C03630=1016.141,-94.892,399.074,165.166,56.508,159.988
C03631=1016.146,-94.643,399.065,165.168,56.502,159.987
C03632=1016.150,-94.393,399.056,165.172,56.496,159.987
C03633=1016.156,-94.143,399.048,165.174,56.489,159.987
C03634=1016.160,-93.893,399.039,165.177,56.484,159.986
C03635=1016.165,-93.643,399.030,165.180,56.477,159.986
C03636=1016.171,-93.394,399.022,165.183,56.472,159.986
C03637=1016.175,-93.144,399.013,165.186,56.465,159.985
C03638=1016.180,-92.894,399.004,165.189,56.459,159.985
C03639=1016.185,-92.644,398.995,165.192,56.453,159.985
C03640=1016.190,-92.394,398.986,165.194,56.446,159.984
C03641=1016.196,-92.144,398.978,165.197,56.441,159.983
C03642=1016.200,-91.894,398.969,165.201,56.434,159.983
C03643=1016.206,-91.645,398.960,165.203,56.428,159.983
C03644=1016.210,-91.395,398.951,165.206,56.422,159.982
C03645=1016.215,-91.145,398.942,165.209,56.416,159.982
C03646=1016.221,-90.896,398.934,165.212,56.409,159.982
C03647=1016.225,-90.646,398.925,165.215,56.403,159.981
C03648=1016.230,-90.396,398.916,165.218,56.397,159.981
C03649=1016.235,-90.146,398.907,165.221,56.391,159.980
C03650=1016.240,-89.896,398.899,165.224,56.385,159.980
C03651=1016.246,-89.647,398.889,165.227,56.379,159.980
C03652=1016.250,-89.397,398.880,165.230,56.372,159.979
C03653=1016.256,-89.147,398.872,165.233,56.366,159.979
C03654=1016.260,-88.897,398.863,165.236,56.359,159.978
///RCONF 1,0,0,0,0,0,0,0,0,0,0,0,0,0,0,0,0,0,0,0,0,0,0,0
C03655=1016.266,-88.647,398.854,165.238,56.354,159.978
C03656=1016.272,-88.398,398.845,165.242,56.347,159.978
C03657=1016.276,-88.148,398.836,165.244,56.341,159.977
C03658=1016.281,-87.898,398.827,165.248,56.335,159.977
C03659=1016.286,-87.648,398.818,165.250,56.328,159.976
C03660=1016.291,-87.398,398.809,165.254,56.322,159.976
C03661=1016.296,-87.149,398.800,165.256,56.316,159.975
C03662=1016.301,-86.899,398.791,165.259,56.309,159.975
C03663=1016.307,-86.650,398.783,165.261,56.303,159.975
C03664=1016.312,-86.399,398.773,165.265,56.297,159.974
C03665=1016.317,-86.120,398.763,165.268,56.290,159.974
C03666=1016.324,-85.839,398.753,165.271,56.283,159.973
C03667=1016.329,-85.559,398.743,165.274,56.275,159.973
C03668=1016.334,-85.278,398.733,165.278,56.268,159.972
C03669=1016.340,-85.029,398.724,165.281,56.262,159.972
C03670=1016.345,-84.779,398.714,165.284,56.256,159.972
C03671=1016.350,-84.530,398.706,165.287,56.250,159.971
C03672=1016.355,-84.280,398.697,165.290,56.243,159.971
C03673=1016.361,-84.030,398.687,165.293,56.237,159.970
C03674=1016.366,-83.780,398.679,165.296,56.230,159.970
C03675=1016.370,-83.530,398.670,165.298,56.224,159.969
C03676=1016.376,-83.281,398.661,165.301,56.218,159.969
C03677=1016.381,-83.031,398.652,165.305,56.211,159.969
C03678=1016.386,-82.780,398.643,165.307,56.205,159.968
C03679=1016.392,-82.531,398.633,165.310,56.198,159.968
C03680=1016.396,-82.281,398.624,165.313,56.193,159.967
C03681=1016.402,-82.032,398.615,165.316,56.186,159.967
C03682=1016.407,-81.782,398.606,165.319,56.179,159.966
C03683=1016.412,-81.532,398.597,165.322,56.173,159.966
C03684=1016.417,-81.282,398.587,165.325,56.166,159.965
C03685=1016.422,-81.033,398.579,165.328,56.160,159.965
C03686=1016.429,-80.783,398.569,165.331,56.154,159.965
C03687=1016.433,-80.533,398.560,165.334,56.147,159.964
C03688=1016.438,-80.283,398.552,165.337,56.141,159.964
C03689=1016.443,-80.034,398.542,165.340,56.134,159.963
C03690=1016.449,-79.784,398.532,165.343,56.128,159.963
C03691=1016.454,-79.534,398.523,165.346,56.122,159.962
C03692=1016.459,-79.285,398.514,165.348,56.116,159.962
C03693=1016.464,-79.034,398.504,165.352,56.109,159.962
C03694=1016.469,-78.784,398.494,165.354,56.103,159.961
C03695=1016.474,-78.535,398.485,165.357,56.096,159.961
C03696=1016.479,-78.285,398.476,165.360,56.091,159.960
C03697=1016.484,-78.035,398.466,165.364,56.085,159.960
C03698=1016.490,-77.786,398.457,165.366,56.078,159.959
C03699=1016.494,-77.536,398.448,165.370,56.072,159.959
C03700=1016.500,-77.286,398.437,165.372,56.066,159.959
C03701=1016.505,-77.037,398.428,165.375,56.059,159.958
C03702=1016.510,-76.787,398.419,165.378,56.053,159.958
C03703=1016.515,-76.537,398.409,165.381,56.046,159.957
C03704=1016.520,-76.287,398.399,165.383,56.040,159.957
C03705=1016.525,-76.038,398.391,165.387,56.034,159.956
C03706=1016.531,-75.787,398.381,165.389,56.028,159.956
C03707=1016.536,-75.538,398.371,165.392,56.021,159.955
C03708=1016.541,-75.287,398.361,165.395,56.015,159.955
C03709=1016.546,-75.038,398.352,165.398,56.008,159.955
C03710=1016.551,-74.789,398.342,165.401,56.003,159.954
C03711=1016.557,-74.539,398.332,165.404,55.996,159.954
C03712=1016.561,-74.289,398.323,165.407,55.990,159.953
C03713=1016.567,-74.039,398.313,165.410,55.983,159.953
C03714=1016.571,-73.789,398.303,165.413,55.978,159.952
C03715=1016.576,-73.540,398.293,165.416,55.972,159.952
C03716=1016.582,-73.290,398.283,165.418,55.965,159.952
C03717=1016.587,-73.040,398.273,165.421,55.959,159.951
C03718=1016.592,-72.790,398.263,165.424,55.953,159.951
C03719=1016.597,-72.541,398.253,165.427,55.947,159.950
C03720=1016.602,-72.291,398.243,165.431,55.941,159.950
C03721=1016.607,-72.041,398.233,165.433,55.934,159.949
C03722=1016.612,-71.792,398.224,165.436,55.929,159.949
C03723=1016.617,-71.542,398.213,165.439,55.922,159.949
C03724=1016.622,-71.292,398.204,165.441,55.916,159.948
C03725=1016.628,-71.042,398.194,165.445,55.910,159.948
C03726=1016.632,-70.793,398.184,165.447,55.904,159.947
C03727=1016.638,-70.543,398.174,165.451,55.897,159.947
C03728=1016.643,-70.293,398.164,165.453,55.891,159.946
C03729=1016.649,-70.015,398.153,165.456,55.884,159.946
C03730=1016.654,-69.737,398.141,165.460,55.877,159.945
C03731=1016.660,-69.458,398.130,165.463,55.870,159.945
C03732=1016.665,-69.180,398.120,165.466,55.864,159.944
C03733=1016.671,-68.930,398.110,165.469,55.857,159.944
C03734=1016.676,-68.681,398.100,165.472,55.851,159.944
C03735=1016.681,-68.430,398.090,165.475,55.844,159.943
C03736=1016.686,-68.181,398.080,165.478,55.839,159.943
C03737=1016.692,-67.932,398.069,165.481,55.832,159.942
C03738=1016.697,-67.681,398.059,165.484,55.826,159.942
C03739=1016.702,-67.432,398.049,165.487,55.819,159.941
C03740=1016.707,-67.182,398.039,165.489,55.814,159.941
C03741=1016.712,-66.933,398.029,165.493,55.807,159.941
C03742=1016.717,-66.682,398.018,165.495,55.801,159.940
C03743=1016.722,-66.433,398.008,165.499,55.794,159.940
C03744=1016.727,-66.183,397.998,165.501,55.788,159.939
C03745=1016.732,-65.933,397.988,165.504,55.782,159.939
C03746=1016.738,-65.684,397.978,165.507,55.775,159.938
C03747=1016.743,-65.434,397.967,165.510,55.769,159.938
C03748=1016.748,-65.184,397.958,165.512,55.763,159.937
C03749=1016.753,-64.934,397.947,165.516,55.756,159.937
C03750=1016.758,-64.685,397.938,165.518,55.750,159.936
C03751=1016.764,-64.435,397.928,165.522,55.744,159.936
C03752=1016.769,-64.185,397.917,165.524,55.738,159.935
C03753=1016.774,-63.936,397.907,165.527,55.731,159.935
C03754=1016.780,-63.686,397.897,165.530,55.725,159.934
C03755=1016.784,-63.436,397.887,165.533,55.719,159.934
C03756=1016.790,-63.186,397.877,165.537,55.712,159.934
C03757=1016.796,-62.937,397.866,165.539,55.705,159.933
C03758=1016.800,-62.687,397.856,165.543,55.699,159.933
C03759=1016.806,-62.437,397.846,165.545,55.693,159.932
C03760=1016.811,-62.187,397.836,165.548,55.686,159.932
C03761=1016.816,-61.938,397.825,165.551,55.680,159.931
C03762=1016.822,-61.688,397.815,165.554,55.674,159.931
C03763=1016.827,-61.438,397.805,165.556,55.667,159.930
C03764=1016.831,-61.188,397.795,165.560,55.661,159.930
C03765=1016.837,-60.939,397.784,165.562,55.655,159.929
C03766=1016.843,-60.689,397.773,165.565,55.648,159.929
C03767=1016.847,-60.439,397.764,165.568,55.641,159.928
C03768=1016.853,-60.190,397.753,165.571,55.635,159.928
C03769=1016.859,-59.940,397.743,165.574,55.629,159.927
C03770=1016.863,-59.690,397.733,165.576,55.622,159.927
C03771=1016.869,-59.440,397.723,165.580,55.615,159.926
C03772=1016.875,-59.191,397.712,165.582,55.610,159.926
C03773=1016.880,-58.940,397.702,165.586,55.603,159.925
C03774=1016.885,-58.691,397.692,165.589,55.596,159.925
C03775=1016.891,-58.442,397.681,165.591,55.590,159.924
C03776=1016.896,-58.191,397.671,165.595,55.584,159.924
C03777=1016.902,-57.942,397.660,165.597,55.577,159.923
C03778=1016.907,-57.693,397.650,165.600,55.570,159.923
C03779=1016.912,-57.442,397.640,165.603,55.564,159.922
C03780=1016.918,-57.193,397.629,165.606,55.557,159.922
C03781=1016.922,-56.943,397.618,165.609,55.550,159.921
C03782=1016.928,-56.694,397.608,165.612,55.545,159.921
C03783=1016.933,-56.444,397.598,165.615,55.538,159.920
C03784=1016.938,-56.194,397.588,165.618,55.531,159.920
C03785=1016.944,-55.944,397.577,165.620,55.525,159.919
C03786=1016.950,-55.694,397.566,165.623,55.518,159.919
C03787=1016.955,-55.445,397.556,165.626,55.512,159.918
C03788=1016.960,-55.195,397.546,165.629,55.506,159.918
C03789=1016.966,-54.946,397.535,165.633,55.499,159.917
C03790=1016.971,-54.695,397.525,165.635,55.492,159.917
C03791=1016.977,-54.445,397.515,165.638,55.486,159.916
C03792=1016.982,-54.197,397.504,165.640,55.479,159.915
C03793=1016.988,-53.919,397.492,165.644,55.471,159.915
C03794=1016.995,-53.642,397.480,165.647,55.465,159.914
C03795=1017.000,-53.365,397.469,165.650,55.457,159.914
C03796=1017.006,-53.088,397.457,165.654,55.450,159.913
C03797=1017.012,-52.838,397.447,165.657,55.444,159.913
C03798=1017.017,-52.588,397.436,165.660,55.437,159.912
C03799=1017.022,-52.338,397.425,165.662,55.430,159.912
C03800=1017.027,-52.089,397.415,165.665,55.424,159.911
C03801=1017.033,-51.839,397.404,165.668,55.417,159.911
C03802=1017.038,-51.589,397.394,165.671,55.410,159.910
C03803=1017.044,-51.340,397.383,165.674,55.404,159.909
C03804=1017.050,-51.090,397.373,165.677,55.397,159.909
C03805=1017.055,-50.840,397.362,165.679,55.391,159.908
C03806=1017.060,-50.590,397.351,165.683,55.384,159.908
C03807=1017.065,-50.340,397.339,165.685,55.378,159.907
C03808=1017.071,-50.090,397.329,165.689,55.371,159.907
C03809=1017.076,-49.841,397.318,165.691,55.366,159.906
C03810=1017.081,-49.591,397.307,165.695,55.359,159.906
C03811=1017.086,-49.341,397.295,165.697,55.353,159.905
C03812=1017.092,-49.091,397.285,165.701,55.347,159.905
C03813=1017.097,-48.842,397.275,165.703,55.340,159.904
C03814=1017.102,-48.593,397.263,165.705,55.334,159.904
C03815=1017.108,-48.343,397.252,165.708,55.327,159.903
C03816=1017.113,-48.093,397.241,165.711,55.321,159.903
C03817=1017.119,-47.844,397.230,165.714,55.315,159.902
C03818=1017.123,-47.593,397.219,165.716,55.308,159.902
C03819=1017.129,-47.344,397.208,165.720,55.302,159.901
C03820=1017.134,-47.094,397.197,165.722,55.296,159.901
C03821=1017.140,-46.845,397.186,165.726,55.289,159.900
C03822=1017.145,-46.595,397.174,165.728,55.283,159.900
C03823=1017.150,-46.345,397.163,165.731,55.276,159.899
C03824=1017.155,-46.095,397.152,165.734,55.270,159.899
C03825=1017.161,-45.846,397.141,165.737,55.264,159.898
C03826=1017.166,-45.596,397.130,165.739,55.257,159.898
C03827=1017.172,-45.347,397.119,165.743,55.251,159.897
C03828=1017.177,-45.096,397.108,165.746,55.244,159.897
C03829=1017.182,-44.847,397.097,165.749,55.238,159.896
C03830=1017.187,-44.597,397.086,165.752,55.231,159.896
C03831=1017.193,-44.347,397.075,165.754,55.225,159.895
C03832=1017.198,-44.098,397.063,165.757,55.218,159.895
C03833=1017.204,-43.848,397.052,165.760,55.212,159.894
C03834=1017.209,-43.598,397.041,165.763,55.205,159.893
C03835=1017.215,-43.349,397.030,165.765,55.199,159.893
C03836=1017.220,-43.099,397.019,165.769,55.193,159.893
C03837=1017.225,-42.850,397.008,165.771,55.186,159.892
C03838=1017.230,-42.600,396.996,165.775,55.180,159.891
C03839=1017.236,-42.350,396.985,165.777,55.173,159.891
C03840=1017.241,-42.101,396.974,165.780,55.167,159.890
C03841=1017.247,-41.850,396.963,165.782,55.160,159.890
C03842=1017.252,-41.601,396.951,165.786,55.154,159.889
C03843=1017.258,-41.351,396.940,165.789,55.147,159.889
C03844=1017.263,-41.101,396.929,165.791,55.140,159.888
C03845=1017.269,-40.852,396.918,165.794,55.134,159.887
C03846=1017.274,-40.602,396.907,165.797,55.128,159.887
C03847=1017.280,-40.352,396.896,165.800,55.121,159.887
C03848=1017.285,-40.103,396.884,165.803,55.115,159.886
C03849=1017.291,-39.854,396.873,165.806,55.108,159.885
C03850=1017.296,-39.604,396.861,165.809,55.102,159.885
C03851=1017.301,-39.353,396.849,165.811,55.095,159.884
C03852=1017.307,-39.104,396.838,165.815,55.088,159.884
C03853=1017.312,-38.854,396.827,165.817,55.082,159.883
C03854=1017.317,-38.604,396.815,165.820,55.077,159.883
C03855=1017.322,-38.355,396.803,165.823,55.070,159.882
C03856=1017.328,-38.106,396.792,165.825,55.063,159.881
C03857=1017.334,-37.828,396.779,165.829,55.057,159.881
C03858=1017.339,-37.551,396.767,165.831,55.049,159.880
C03859=1017.346,-37.275,396.754,165.835,55.043,159.880
C03860=1017.351,-36.998,396.741,165.838,55.035,159.879
C03861=1017.356,-36.748,396.730,165.841,55.028,159.879
C03862=1017.362,-36.499,396.717,165.843,55.023,159.878
C03863=1017.368,-36.249,396.706,165.847,55.016,159.878
C03864=1017.373,-35.999,396.695,165.849,55.010,159.877
C03865=1017.378,-35.750,396.682,165.852,55.003,159.876
C03866=1017.383,-35.500,396.671,165.855,54.997,159.876
C03867=1017.389,-35.250,396.659,165.858,54.990,159.875
C03868=1017.395,-35.001,396.648,165.860,54.984,159.875
C03869=1017.400,-34.751,396.636,165.864,54.978,159.874
C03870=1017.405,-34.501,396.625,165.866,54.971,159.874
C03871=1017.410,-34.252,396.612,165.870,54.965,159.873
C03872=1017.416,-34.002,396.601,165.872,54.958,159.873
C03873=1017.422,-33.752,396.590,165.875,54.952,159.872
C03874=1017.427,-33.503,396.578,165.877,54.945,159.871
C03875=1017.432,-33.253,396.566,165.881,54.939,159.871
C03876=1017.438,-33.003,396.554,165.883,54.932,159.870
C03877=1017.443,-32.753,396.542,165.886,54.925,159.870
C03878=1017.449,-32.504,396.531,165.888,54.919,159.869
C03879=1017.454,-32.255,396.519,165.892,54.912,159.869
C03880=1017.459,-32.004,396.507,165.895,54.907,159.868
C03881=1017.465,-31.755,396.495,165.898,54.900,159.868
C03882=1017.470,-31.505,396.483,165.900,54.894,159.867
C03883=1017.476,-31.256,396.472,165.903,54.887,159.867
C03884=1017.481,-31.006,396.460,165.906,54.881,159.866
C03885=1017.486,-30.756,396.449,165.909,54.874,159.865
C03886=1017.492,-30.507,396.436,165.911,54.868,159.865
C03887=1017.497,-30.256,396.425,165.915,54.861,159.864
C03888=1017.503,-30.008,396.413,165.917,54.855,159.864
C03889=1017.508,-29.758,396.401,165.920,54.848,159.863
C03890=1017.514,-29.508,396.389,165.923,54.842,159.862
C03891=1017.519,-29.258,396.377,165.926,54.835,159.862
C03892=1017.525,-29.009,396.365,165.928,54.829,159.861
C03893=1017.531,-28.759,396.354,165.931,54.822,159.861
C03894=1017.536,-28.510,396.342,165.935,54.815,159.860
C03895=1017.541,-28.260,396.330,165.937,54.809,159.860
C03896=1017.547,-28.010,396.318,165.940,54.802,159.859
C03897=1017.552,-27.760,396.306,165.942,54.795,159.858
C03898=1017.557,-27.511,396.294,165.946,54.789,159.858
C03899=1017.563,-27.261,396.282,165.948,54.783,159.857
C03900=1017.568,-27.011,396.270,165.951,54.777,159.857
C03901=1017.574,-26.762,396.258,165.954,54.770,159.856
C03902=1017.580,-26.512,396.245,165.956,54.764,159.855
C03903=1017.585,-26.262,396.234,165.959,54.757,159.855
C03904=1017.591,-26.012,396.221,165.962,54.751,159.854
C03905=1017.596,-25.763,396.209,165.965,54.744,159.854
C03906=1017.601,-25.514,396.197,165.968,54.739,159.853
C03907=1017.607,-25.264,396.185,165.970,54.732,159.853
C03908=1017.611,-25.014,396.172,165.973,54.726,159.852
C03909=1017.617,-24.764,396.160,165.976,54.719,159.852
C03910=1017.623,-24.515,396.148,165.979,54.713,159.851
C03911=1017.628,-24.265,396.136,165.981,54.706,159.850
C03912=1017.633,-24.015,396.124,165.985,54.700,159.850
C03913=1017.639,-23.766,396.111,165.987,54.693,159.849
C03914=1017.645,-23.516,396.099,165.989,54.687,159.849
C03915=1017.650,-23.266,396.087,165.993,54.680,159.848
C03916=1017.655,-23.017,396.075,165.995,54.674,159.847
C03917=1017.661,-22.767,396.063,165.998,54.667,159.847
C03918=1017.666,-22.518,396.050,166.001,54.661,159.846
C03919=1017.671,-22.268,396.037,166.004,54.654,159.846
C03920=1017.676,-22.018,396.026,166.006,54.648,159.845
C03921=1017.683,-21.741,396.012,166.010,54.641,159.845
C03922=1017.689,-21.463,395.999,166.012,54.634,159.844
C03923=1017.695,-21.185,395.985,166.015,54.627,159.843
C03924=1017.701,-20.907,395.971,166.019,54.620,159.843
C03925=1017.707,-20.658,395.959,166.022,54.613,159.842
C03926=1017.713,-20.408,395.946,166.024,54.606,159.841
C03927=1017.718,-20.158,395.935,166.027,54.600,159.841
C03928=1017.724,-19.908,395.922,166.029,54.593,159.840
C03929=1017.728,-19.659,395.909,166.033,54.587,159.840
C03930=1017.734,-19.409,395.897,166.035,54.580,159.839
C03931=1017.739,-19.160,395.884,166.038,54.574,159.838
C03932=1017.745,-18.910,395.872,166.041,54.567,159.838
C03933=1017.751,-18.661,395.860,166.044,54.561,159.837
C03934=1017.756,-18.411,395.847,166.046,54.555,159.837
C03935=1017.762,-18.162,395.835,166.050,54.548,159.836
C03936=1017.768,-17.912,395.822,166.052,54.542,159.835
C03937=1017.773,-17.663,395.810,166.055,54.535,159.835
C03938=1017.778,-17.412,395.798,166.058,54.529,159.834
C03939=1017.783,-17.163,395.786,166.061,54.522,159.834
C03940=1017.789,-16.913,395.773,166.063,54.515,159.833
C03941=1017.795,-16.663,395.760,166.066,54.508,159.832
C03942=1017.800,-16.414,395.748,166.069,54.502,159.832
C03943=1017.806,-16.164,395.736,166.072,54.495,159.831
C03944=1017.811,-15.915,395.724,166.074,54.489,159.830
C03945=1017.817,-15.665,395.710,166.078,54.482,159.830
C03946=1017.822,-15.416,395.698,166.080,54.476,159.829
C03947=1017.828,-15.166,395.685,166.082,54.470,159.829
C03948=1017.833,-14.917,395.672,166.086,54.463,159.828
C03949=1017.839,-14.667,395.660,166.088,54.457,159.827
C03950=1017.844,-14.417,395.646,166.090,54.451,159.827
C03951=1017.849,-14.167,395.634,166.094,54.444,159.826
C03952=1017.855,-13.917,395.622,166.096,54.438,159.826
C03953=1017.860,-13.669,395.608,166.099,54.431,159.825
C03954=1017.866,-13.419,395.596,166.102,54.425,159.824
C03955=1017.871,-13.168,395.583,166.104,54.419,159.824
C03956=1017.876,-12.919,395.570,166.107,54.412,159.823
C03957=1017.882,-12.669,395.558,166.110,54.406,159.823
C03958=1017.888,-12.420,395.544,166.113,54.399,159.822
C03959=1017.893,-12.171,395.532,166.115,54.393,159.821
C03960=1017.898,-11.920,395.519,166.118,54.387,159.821
C03961=1017.903,-11.671,395.506,166.121,54.380,159.820
C03962=1017.909,-11.421,395.494,166.123,54.374,159.820
C03963=1017.915,-11.172,395.480,166.127,54.367,159.819
C03964=1017.920,-10.923,395.468,166.129,54.361,159.818
C03965=1017.926,-10.673,395.455,166.132,54.355,159.818
C03966=1017.931,-10.423,395.442,166.135,54.348,159.817
C03967=1017.937,-10.174,395.429,166.137,54.342,159.817
C03968=1017.942,-9.924,395.416,166.141,54.335,159.816
C03969=1017.948,-9.674,395.403,166.143,54.329,159.815
C03970=1017.954,-9.425,395.391,166.146,54.321,159.815
C03971=1017.959,-9.175,395.377,166.148,54.315,159.814
C03972=1017.965,-8.925,395.365,166.151,54.309,159.813
C03973=1017.969,-8.676,395.352,166.154,54.302,159.813
C03974=1017.975,-8.427,395.339,166.156,54.296,159.812
C03975=1017.981,-8.177,395.326,166.160,54.289,159.812
C03976=1017.986,-7.926,395.313,166.162,54.283,159.811
C03977=1017.992,-7.678,395.300,166.165,54.277,159.811
C03978=1017.997,-7.428,395.287,166.167,54.270,159.810
C03979=1018.003,-7.178,395.275,166.171,54.263,159.809
C03980=1018.009,-6.929,395.262,166.173,54.257,159.808
C03981=1018.014,-6.679,395.248,166.175,54.251,159.808
C03982=1018.020,-6.429,395.236,166.179,54.244,159.807
C03983=1018.025,-6.180,395.222,166.181,54.238,159.807
C03984=1018.031,-5.930,395.210,166.184,54.230,159.806
C03985=1018.038,-5.650,395.195,166.187,54.223,159.805
C03986=1018.043,-5.371,395.180,166.190,54.216,159.804
C03987=1018.050,-5.091,395.166,166.193,54.209,159.804
C03988=1018.056,-4.812,395.151,166.196,54.202,159.803
C03989=1018.062,-4.562,395.138,166.199,54.194,159.802
C03990=1018.067,-4.313,395.125,166.201,54.188,159.802
C03991=1018.072,-4.063,395.112,166.204,54.182,159.801
C03992=1018.078,-3.813,395.098,166.207,54.175,159.801
C03993=1018.083,-3.563,395.085,166.210,54.169,159.800
C03994=1018.089,-3.314,395.072,166.212,54.163,159.799
C03995=1018.094,-3.064,395.059,166.215,54.156,159.799
C03996=1018.099,-2.815,395.045,166.218,54.150,159.798
C03997=1018.105,-2.565,395.031,166.220,54.144,159.797
C03998=1018.111,-2.315,395.019,166.223,54.137,159.797
C03999=1018.116,-2.066,395.005,166.226,54.131,159.796
C04000=1018.121,-1.817,394.991,166.228,54.125,159.796
C04001=1018.126,-1.567,394.978,166.232,54.118,159.795
C04002=1018.132,-1.317,394.964,166.234,54.112,159.794
C04003=1018.138,-1.068,394.951,166.236,54.106,159.794
C04004=1018.143,-0.818,394.938,166.239,54.099,159.793
C04005=1018.148,-0.569,394.924,166.242,54.093,159.793
C04006=1018.153,-0.319,394.911,166.244,54.087,159.792
C04007=1018.159,-0.069,394.898,166.247,54.080,159.791
C04008=1018.165,0.180,394.884,166.250,54.074,159.791
C04009=1018.170,0.430,394.870,166.253,54.068,159.790
C04010=1018.175,0.680,394.857,166.255,54.061,159.789
C04011=1018.180,0.929,394.844,166.258,54.055,159.789
C04012=1018.186,1.178,394.830,166.261,54.049,159.788
C04013=1018.192,1.428,394.817,166.263,54.042,159.788
C04014=1018.197,1.678,394.803,166.266,54.035,159.787
C04015=1018.203,1.927,394.789,166.268,54.029,159.786
C04016=1018.209,2.177,394.776,166.272,54.022,159.786
C04017=1018.214,2.426,394.762,166.274,54.016,159.785
C04018=1018.219,2.676,394.749,166.277,54.010,159.784
C04019=1018.224,2.925,394.736,166.280,54.003,159.784
C04020=1018.230,3.175,394.722,166.282,53.997,159.783
C04021=1018.236,3.424,394.709,166.285,53.991,159.783
C04022=1018.241,3.674,394.695,166.288,53.983,159.782
C04023=1018.247,3.924,394.682,166.290,53.977,159.781
C04024=1018.252,4.174,394.668,166.292,53.971,159.780
C04025=1018.258,4.423,394.654,166.296,53.964,159.780
C04026=1018.264,4.672,394.641,166.298,53.958,159.779
C04027=1018.269,4.922,394.627,166.301,53.952,159.779
C04028=1018.274,5.172,394.614,166.304,53.945,159.778
C04029=1018.280,5.422,394.600,166.306,53.939,159.777
C04030=1018.286,5.671,394.586,166.309,53.932,159.777
C04031=1018.292,5.921,394.573,166.312,53.926,159.776
C04032=1018.297,6.169,394.559,166.314,53.920,159.775
C04033=1018.302,6.419,394.545,166.317,53.912,159.775
C04034=1018.307,6.669,394.532,166.320,53.906,159.774
C04035=1018.313,6.918,394.519,166.322,53.900,159.773
C04036=1018.319,7.168,394.505,166.325,53.893,159.773
C04037=1018.324,7.418,394.491,166.327,53.886,159.772
C04038=1018.330,7.667,394.477,166.331,53.880,159.771
C04039=1018.335,7.917,394.463,166.333,53.874,159.771
C04040=1018.342,8.166,394.450,166.336,53.867,159.770
C04041=1018.347,8.416,394.436,166.339,53.860,159.769
C04042=1018.352,8.665,394.422,166.341,53.854,159.769
C04043=1018.358,8.915,394.408,166.344,53.847,159.768
C04044=1018.363,9.165,394.395,166.347,53.841,159.767
C04045=1018.369,9.414,394.382,166.349,53.834,159.767
C04046=1018.375,9.664,394.368,166.352,53.828,159.766
C04047=1018.380,9.913,394.354,166.355,53.821,159.765
C04048=1018.386,10.163,394.340,166.358,53.814,159.765
C04049=1018.393,10.444,394.325,166.361,53.807,159.764
C04050=1018.399,10.726,394.309,166.363,53.800,159.763
C04051=1018.405,11.008,394.294,166.366,53.792,159.762
C04052=1018.411,11.289,394.278,166.369,53.785,159.762
C04053=1018.418,11.538,394.264,166.371,53.778,159.761
C04054=1018.423,11.788,394.251,166.375,53.772,159.760
C04055=1018.429,12.038,394.237,166.377,53.765,159.760
C04056=1018.434,12.287,394.223,166.380,53.758,159.759
C04057=1018.440,12.550,394.209,166.383,53.752,159.758
C04058=1018.446,12.813,394.194,166.386,53.745,159.757
C04059=1018.452,13.076,394.180,166.389,53.737,159.757
C04060=1018.458,13.339,394.165,166.391,53.731,159.756
C04061=1018.463,13.588,394.151,166.394,53.724,159.755
C04062=1018.469,13.838,394.137,166.396,53.718,159.755
C04063=1018.474,14.087,394.122,166.399,53.712,159.754
C04064=1018.480,14.336,394.109,166.402,53.705,159.753
C04065=1018.485,14.586,394.095,166.405,53.699,159.753
C04066=1018.491,14.836,394.081,166.407,53.692,159.752
C04067=1018.496,15.085,394.067,166.410,53.685,159.751
C04068=1018.502,15.335,394.051,166.413,53.679,159.751
C04069=1018.508,15.585,394.038,166.415,53.673,159.750
C04070=1018.513,15.834,394.024,166.418,53.666,159.749
C04071=1018.518,16.084,394.010,166.420,53.660,159.749
C04072=1018.524,16.333,393.995,166.423,53.654,159.748
C04073=1018.530,16.582,393.981,166.425,53.647,159.747
C04074=1018.535,16.832,393.968,166.428,53.640,159.746
C04075=1018.541,17.082,393.954,166.431,53.634,159.746
C04076=1018.546,17.331,393.939,166.433,53.628,159.745
C04077=1018.553,17.581,393.925,166.437,53.621,159.745
C04078=1018.557,17.831,393.910,166.439,53.614,159.744
C04079=1018.563,18.080,393.897,166.441,53.608,159.743
C04080=1018.569,18.329,393.882,166.444,53.602,159.743
C04081=1018.574,18.579,393.868,166.446,53.595,159.742
C04082=1018.579,18.828,393.854,166.450,53.588,159.741
C04083=1018.586,19.078,393.839,166.452,53.582,159.741
C04084=1018.591,19.328,393.825,166.455,53.576,159.740
C04085=1018.596,19.578,393.811,166.457,53.569,159.739
C04086=1018.602,19.826,393.796,166.460,53.562,159.738
C04087=1018.607,20.076,393.783,166.463,53.556,159.738
C04088=1018.613,20.325,393.768,166.465,53.550,159.737
C04089=1018.618,20.576,393.753,166.468,53.543,159.736
C04090=1018.624,20.825,393.739,166.471,53.537,159.736
C04091=1018.630,21.074,393.725,166.473,53.531,159.735
C04092=1018.635,21.324,393.711,166.475,53.524,159.734
C04093=1018.640,21.573,393.696,166.478,53.517,159.734
C04094=1018.646,21.823,393.681,166.481,53.511,159.733
C04095=1018.652,22.072,393.667,166.483,53.505,159.732
C04096=1018.658,22.322,393.653,166.487,53.498,159.732
C04097=1018.662,22.572,393.639,166.489,53.492,159.731
C04098=1018.668,22.821,393.624,166.491,53.485,159.730
C04099=1018.674,23.071,393.610,166.495,53.479,159.730
C04100=1018.680,23.320,393.595,166.497,53.472,159.729
C04101=1018.685,23.570,393.581,166.499,53.466,159.728
C04102=1018.690,23.819,393.566,166.503,53.459,159.728
C04103=1018.697,24.069,393.552,166.505,53.452,159.727
C04104=1018.702,24.318,393.537,166.507,53.446,159.726
C04105=1018.707,24.568,393.523,166.511,53.440,159.726
C04106=1018.713,24.817,393.508,166.513,53.433,159.725
C04107=1018.719,25.067,393.494,166.515,53.427,159.724
C04108=1018.724,25.316,393.479,166.519,53.420,159.723
C04109=1018.729,25.566,393.465,166.521,53.413,159.723
C04110=1018.735,25.815,393.450,166.523,53.407,159.722
C04111=1018.742,26.064,393.435,166.525,53.401,159.721
C04112=1018.746,26.314,393.421,166.528,53.394,159.721
C04113=1018.752,26.584,393.405,166.532,53.387,159.720
C04114=1018.759,26.854,393.389,166.534,53.381,159.719
C04115=1018.765,27.123,393.374,166.537,53.373,159.718
C04116=1018.771,27.394,393.358,166.540,53.366,159.718
C04117=1018.776,27.643,393.343,166.542,53.359,159.717
C04118=1018.782,27.892,393.329,166.545,53.353,159.716
C04119=1018.787,28.143,393.314,166.548,53.347,159.716
C04120=1018.793,28.392,393.299,166.550,53.341,159.715
C04121=1018.798,28.641,393.284,166.553,53.334,159.714
C04122=1018.804,28.891,393.269,166.555,53.328,159.713
C04123=1018.809,29.140,393.255,166.558,53.321,159.713
C04124=1018.815,29.389,393.240,166.561,53.315,159.712
C04125=1018.820,29.639,393.224,166.563,53.308,159.711
C04126=1018.826,29.888,393.210,166.565,53.302,159.711
C04127=1018.831,30.138,393.195,166.569,53.295,159.710
C04128=1018.837,30.388,393.181,166.571,53.289,159.709
C04129=1018.842,30.637,393.165,166.573,53.282,159.708
C04130=1018.848,30.886,393.151,166.576,53.276,159.708
C04131=1018.853,31.137,393.136,166.579,53.269,159.707
C04132=1018.859,31.386,393.121,166.581,53.263,159.706
C04133=1018.864,31.635,393.106,166.584,53.257,159.706
C04134=1018.871,31.885,393.091,166.587,53.250,159.705
C04135=1018.876,32.134,393.076,166.589,53.244,159.704
C04136=1018.881,32.383,393.062,166.592,53.237,159.704
C04137=1018.887,32.633,393.047,166.594,53.231,159.703
C04138=1018.893,32.882,393.032,166.597,53.224,159.702
C04139=1018.898,33.132,393.017,166.600,53.218,159.702
C04140=1018.903,33.382,393.001,166.602,53.211,159.701
C04141=1018.909,33.631,392.987,166.605,53.205,159.700
C04142=1018.914,33.881,392.972,166.608,53.198,159.699
C04143=1018.920,34.130,392.957,166.610,53.192,159.699
C04144=1018.925,34.379,392.942,166.612,53.186,159.698
C04145=1018.932,34.629,392.927,166.616,53.178,159.697
C04146=1018.937,34.878,392.912,166.618,53.172,159.697
C04147=1018.943,35.128,392.897,166.620,53.166,159.696
C04148=1018.948,35.378,392.883,166.624,53.159,159.695
C04149=1018.954,35.627,392.868,166.626,53.153,159.694
C04150=1018.959,35.877,392.853,166.628,53.146,159.694
C04151=1018.965,36.126,392.838,166.632,53.140,159.693
C04152=1018.971,36.376,392.822,166.634,53.133,159.692
C04153=1018.976,36.625,392.808,166.636,53.127,159.692
C04154=1018.982,36.875,392.792,166.639,53.121,159.691
C04155=1018.987,37.124,392.777,166.642,53.113,159.690
C04156=1018.993,37.374,392.762,166.644,53.107,159.689
C04157=1018.998,37.623,392.746,166.647,53.101,159.689
C04158=1019.004,37.873,392.731,166.649,53.094,159.688
C04159=1019.009,38.122,392.716,166.652,53.088,159.687
C04160=1019.014,38.371,392.701,166.655,53.082,159.687
C04161=1019.020,38.621,392.686,166.657,53.075,159.686
C04162=1019.026,38.870,392.671,166.659,53.069,159.685
C04163=1019.031,39.120,392.655,166.663,53.062,159.685
C04164=1019.036,39.369,392.640,166.665,53.056,159.684
C04165=1019.042,39.619,392.624,166.667,53.050,159.683
C04166=1019.048,39.868,392.609,166.670,53.043,159.682
C04167=1019.054,40.118,392.594,166.673,53.036,159.682
C04168=1019.059,40.367,392.579,166.676,53.030,159.681
C04169=1019.064,40.617,392.563,166.678,53.024,159.680
C04170=1019.070,40.866,392.548,166.680,53.017,159.679
C04171=1019.076,41.116,392.533,166.684,53.011,159.679
C04172=1019.081,41.365,392.518,166.686,53.004,159.678
C04173=1019.087,41.615,392.502,166.688,52.998,159.677
C04174=1019.092,41.864,392.486,166.691,52.992,159.677
C04175=1019.098,42.113,392.472,166.694,52.985,159.676
C04176=1019.103,42.363,392.456,166.696,52.979,159.675
C04177=1019.109,42.646,392.438,166.699,52.971,159.675
C04178=1019.115,42.929,392.421,166.703,52.964,159.674
C04179=1019.122,43.212,392.403,166.705,52.957,159.673
C04180=1019.128,43.495,392.385,166.707,52.950,159.672
C04181=1019.133,43.744,392.370,166.710,52.944,159.671
C04182=1019.139,43.994,392.354,166.713,52.937,159.671
C04183=1019.144,44.243,392.338,166.716,52.931,159.670
C04184=1019.150,44.493,392.323,166.718,52.924,159.669
C04185=1019.155,44.742,392.308,166.721,52.918,159.669
C04186=1019.161,44.992,392.291,166.723,52.912,159.668
C04187=1019.166,45.241,392.276,166.726,52.906,159.667
C04188=1019.171,45.491,392.261,166.729,52.899,159.666
C04189=1019.177,45.740,392.245,166.731,52.893,159.666
C04190=1019.182,45.990,392.229,166.734,52.887,159.665
C04191=1019.188,46.239,392.213,166.736,52.880,159.664
C04192=1019.192,46.488,392.197,166.738,52.874,159.664
C04193=1019.198,46.738,392.182,166.742,52.867,159.663
C04194=1019.203,46.987,392.166,166.744,52.861,159.662
C04195=1019.209,47.237,392.150,166.746,52.854,159.661
C04196=1019.214,47.486,392.134,166.749,52.848,159.661
C04197=1019.220,47.736,392.119,166.751,52.842,159.660
C04198=1019.226,47.986,392.103,166.755,52.835,159.659
C04199=1019.231,48.234,392.087,166.757,52.829,159.659
C04200=1019.237,48.484,392.072,166.759,52.822,159.658
C04201=1019.242,48.733,392.056,166.762,52.816,159.657
C04202=1019.248,48.983,392.040,166.764,52.810,159.657
C04203=1019.254,49.232,392.024,166.767,52.803,159.656
C04204=1019.259,49.481,392.009,166.770,52.797,159.655
C04205=1019.264,49.731,391.993,166.773,52.791,159.654
C04206=1019.269,49.980,391.977,166.775,52.784,159.654
C04207=1019.275,50.230,391.961,166.778,52.778,159.653
C04208=1019.281,50.480,391.945,166.780,52.771,159.652
C04209=1019.286,50.729,391.930,166.783,52.765,159.652
C04210=1019.292,50.978,391.914,166.785,52.758,159.651
C04211=1019.297,51.228,391.898,166.788,52.752,159.650
C04212=1019.303,51.477,391.882,166.791,52.746,159.649
C04213=1019.308,51.727,391.867,166.793,52.739,159.649
C04214=1019.314,51.976,391.850,166.796,52.733,159.648
C04215=1019.319,52.226,391.835,166.798,52.726,159.647
C04216=1019.325,52.475,391.819,166.801,52.720,159.646
C04217=1019.330,52.724,391.804,166.804,52.713,159.646
C04218=1019.335,52.974,391.787,166.806,52.707,159.645
C04219=1019.341,53.224,391.771,166.808,52.700,159.644
C04220=1019.347,53.473,391.755,166.812,52.694,159.644
C04221=1019.352,53.722,391.739,166.814,52.688,159.643
C04222=1019.358,53.972,391.724,166.816,52.681,159.642
C04223=1019.364,54.221,391.707,166.819,52.675,159.641
C04224=1019.369,54.470,391.692,166.822,52.668,159.641
C04225=1019.375,54.720,391.676,166.825,52.662,159.640
C04226=1019.381,54.970,391.660,166.827,52.655,159.639
C04227=1019.386,55.218,391.645,166.830,52.648,159.638
C04228=1019.392,55.468,391.628,166.832,52.642,159.638
C04229=1019.397,55.718,391.612,166.835,52.635,159.637
C04230=1019.403,55.967,391.596,166.837,52.629,159.636
C04231=1019.408,56.217,391.581,166.840,52.622,159.635
C04232=1019.414,56.466,391.565,166.843,52.616,159.635
C04233=1019.420,56.715,391.548,166.845,52.609,159.634
C04234=1019.425,56.964,391.533,166.848,52.603,159.633
C04235=1019.431,57.214,391.517,166.851,52.596,159.632
C04236=1019.437,57.463,391.501,166.853,52.590,159.632
C04237=1019.442,57.713,391.485,166.855,52.583,159.631
C04238=1019.448,57.962,391.469,166.859,52.577,159.630
C04239=1019.453,58.212,391.454,166.861,52.570,159.629
C04240=1019.459,58.461,391.437,166.863,52.563,159.628
C04241=1019.465,58.744,391.418,166.866,52.556,159.628
C04242=1019.472,59.027,391.401,166.869,52.548,159.627
C04243=1019.478,59.311,391.382,166.872,52.541,159.626
C04244=1019.484,59.592,391.364,166.875,52.533,159.625
C04245=1019.490,59.842,391.348,166.879,52.527,159.624
C04246=1019.496,60.092,391.333,166.881,52.520,159.624
C04247=1019.502,60.341,391.316,166.883,52.514,159.623
C04248=1019.507,60.591,391.300,166.887,52.507,159.622
C04249=1019.512,60.840,391.284,166.889,52.500,159.621
C04250=1019.518,61.089,391.268,166.891,52.494,159.621
C04251=1019.524,61.339,391.252,166.894,52.487,159.620
C04252=1019.530,61.588,391.236,166.897,52.480,159.619
C04253=1019.536,61.838,391.220,166.899,52.474,159.618
C04254=1019.541,62.087,391.204,166.902,52.467,159.618
C04255=1019.547,62.336,391.188,166.904,52.461,159.617
C04256=1019.553,62.585,391.172,166.907,52.455,159.616
C04257=1019.558,62.836,391.156,166.910,52.448,159.615
C04258=1019.564,63.085,391.139,166.913,52.442,159.615
C04259=1019.570,63.334,391.123,166.915,52.435,159.614
C04260=1019.575,63.584,391.106,166.918,52.429,159.613
C04261=1019.580,63.833,391.090,166.921,52.422,159.612
C04262=1019.586,64.082,391.073,166.923,52.416,159.612
C04263=1019.591,64.332,391.057,166.925,52.409,159.611
C04264=1019.597,64.581,391.041,166.928,52.402,159.610
C04265=1019.603,64.831,391.024,166.931,52.396,159.609
C04266=1019.609,65.080,391.008,166.933,52.389,159.608
C04267=1019.614,65.330,390.991,166.936,52.383,159.608
C04268=1019.619,65.578,390.975,166.938,52.376,159.607
C04269=1019.624,65.828,390.958,166.942,52.370,159.606
C04270=1019.630,66.077,390.942,166.944,52.363,159.606
C04271=1019.636,66.327,390.926,166.947,52.357,159.605
C04272=1019.641,66.576,390.909,166.949,52.351,159.604
C04273=1019.647,66.826,390.893,166.952,52.344,159.603
C04274=1019.653,67.075,390.876,166.955,52.337,159.603
C04275=1019.658,67.324,390.860,166.957,52.331,159.602
C04276=1019.663,67.574,390.843,166.959,52.325,159.601
C04277=1019.669,67.823,390.827,166.963,52.318,159.601
C04278=1019.674,68.073,390.810,166.965,52.312,159.600
C04279=1019.680,68.322,390.794,166.967,52.305,159.599
C04280=1019.686,68.572,390.777,166.970,52.299,159.598
C04281=1019.691,68.821,390.761,166.973,52.292,159.597
C04282=1019.697,69.071,390.744,166.976,52.286,159.597
C04283=1019.702,69.320,390.727,166.978,52.279,159.596
C04284=1019.708,69.570,390.711,166.980,52.273,159.595
C04285=1019.713,69.818,390.693,166.983,52.266,159.594
C04286=1019.718,70.068,390.677,166.986,52.260,159.594
C04287=1019.724,70.317,390.660,166.988,52.253,159.593
C04288=1019.729,70.567,390.643,166.991,52.247,159.592
C04289=1019.735,70.816,390.627,166.993,52.241,159.591
C04290=1019.740,71.066,390.610,166.997,52.234,159.591
C04291=1019.746,71.315,390.593,166.999,52.228,159.590
C04292=1019.752,71.564,390.576,167.002,52.222,159.589
C04293=1019.757,71.814,390.560,167.004,52.215,159.588
C04294=1019.762,72.063,390.543,167.007,52.209,159.588
C04295=1019.768,72.313,390.527,167.010,52.202,159.587
C04296=1019.774,72.562,390.509,167.012,52.196,159.586
C04297=1019.779,72.811,390.492,167.014,52.189,159.585
C04298=1019.785,73.061,390.476,167.018,52.182,159.585
C04299=1019.790,73.311,390.459,167.020,52.176,159.584
C04300=1019.796,73.560,390.441,167.022,52.170,159.583
C04301=1019.802,73.809,390.425,167.025,52.164,159.582
C04302=1019.806,74.058,390.409,167.028,52.156,159.582
C04303=1019.812,74.307,390.392,167.031,52.150,159.581
C04304=1019.818,74.556,390.375,167.033,52.144,159.580
C04305=1019.824,74.840,390.356,167.036,52.136,159.579
C04306=1019.831,75.123,390.337,167.039,52.129,159.578
C04307=1019.837,75.405,390.318,167.042,52.121,159.577
C04308=1019.843,75.688,390.299,167.045,52.114,159.577
C04309=1019.849,75.937,390.281,167.047,52.108,159.576
C04310=1019.854,76.187,390.264,167.051,52.101,159.575
C04311=1019.860,76.436,390.248,167.053,52.095,159.574
C04312=1019.865,76.685,390.230,167.056,52.089,159.574
C04313=1019.870,76.935,390.214,167.059,52.082,159.573
C04314=1019.876,77.184,390.196,167.061,52.075,159.572
C04315=1019.881,77.434,390.179,167.064,52.069,159.571
C04316=1019.886,77.683,390.162,167.066,52.062,159.571
C04317=1019.892,77.932,390.145,167.069,52.056,159.570
C04318=1019.898,78.182,390.128,167.072,52.049,159.569
C04319=1019.903,78.431,390.111,167.075,52.043,159.568
C04320=1019.909,78.681,390.094,167.077,52.037,159.568
C04321=1019.914,78.930,390.076,167.080,52.031,159.567
C04322=1019.919,79.179,390.060,167.083,52.024,159.566
C04323=1019.925,79.428,390.042,167.085,52.018,159.565
C04324=1019.930,79.678,390.025,167.088,52.011,159.565
C04325=1019.936,79.927,390.008,167.090,52.005,159.564
C04326=1019.941,80.176,389.990,167.093,51.998,159.563
C04327=1019.946,80.426,389.973,167.096,51.992,159.563
C04328=1019.952,80.675,389.956,167.098,51.985,159.562
C04329=1019.957,80.924,389.939,167.101,51.979,159.561
C04330=1019.963,81.173,389.921,167.103,51.973,159.560
C04331=1019.968,81.424,389.904,167.107,51.966,159.559
C04332=1019.974,81.673,389.886,167.109,51.960,159.559
C04333=1019.979,81.922,389.870,167.111,51.953,159.558
C04334=1019.985,82.172,389.852,167.114,51.947,159.557
C04335=1019.990,82.421,389.834,167.117,51.940,159.556
C04336=1019.995,82.670,389.818,167.120,51.933,159.556
C04337=1020.002,82.919,389.801,167.122,51.927,159.555
C04338=1020.007,83.169,389.784,167.125,51.920,159.554
C04339=1020.012,83.418,389.766,167.128,51.914,159.553
C04340=1020.018,83.667,389.749,167.130,51.908,159.553
C04341=1020.024,83.917,389.731,167.133,51.901,159.552
C04342=1020.029,84.166,389.714,167.136,51.895,159.551
C04343=1020.035,84.415,389.696,167.138,51.888,159.550
C04344=1020.040,84.665,389.679,167.141,51.882,159.549
C04345=1020.045,84.914,389.662,167.144,51.875,159.549
C04346=1020.051,85.163,389.644,167.147,51.869,159.548
C04347=1020.056,85.413,389.627,167.149,51.862,159.547
C04348=1020.062,85.662,389.610,167.152,51.856,159.546
C04349=1020.068,85.911,389.592,167.155,51.849,159.546
C04350=1020.073,86.161,389.575,167.157,51.842,159.545
C04351=1020.079,86.410,389.558,167.160,51.836,159.544
C04352=1020.084,86.659,389.540,167.163,51.829,159.543
C04353=1020.089,86.909,389.523,167.165,51.823,159.543
C04354=1020.095,87.158,389.506,167.168,51.817,159.542
C04355=1020.101,87.407,389.488,167.171,51.810,159.541
C04356=1020.106,87.657,389.471,167.173,51.803,159.540
C04357=1020.112,87.906,389.453,167.176,51.797,159.540
C04358=1020.117,88.155,389.436,167.179,51.790,159.539
C04359=1020.123,88.404,389.418,167.182,51.784,159.538
C04360=1020.128,88.654,389.401,167.184,51.777,159.537
C04361=1020.134,88.904,389.383,167.188,51.771,159.537
C04362=1020.140,89.153,389.366,167.190,51.764,159.536
C04363=1020.145,89.402,389.348,167.192,51.757,159.535
C04364=1020.151,89.651,389.331,167.195,51.751,159.534
C04365=1020.156,89.901,389.313,167.198,51.744,159.533
C04366=1020.161,90.151,389.295,167.201,51.739,159.533
C04367=1020.167,90.400,389.278,167.203,51.732,159.532
C04368=1020.172,90.649,389.260,167.206,51.726,159.531
C04369=1020.178,90.931,389.240,167.209,51.718,159.530
C04370=1020.184,91.214,389.219,167.212,51.711,159.529
C04371=1020.190,91.497,389.199,167.215,51.704,159.528
C04372=1020.197,91.780,389.179,167.218,51.697,159.528
C04373=1020.202,92.030,389.161,167.221,51.690,159.527
C04374=1020.207,92.279,389.144,167.224,51.684,159.526
C04375=1020.213,92.528,389.126,167.226,51.677,159.525
C04376=1020.219,92.778,389.108,167.228,51.671,159.525
C04377=1020.224,93.027,389.090,167.232,51.664,159.524
C04378=1020.229,93.276,389.073,167.234,51.658,159.523
C04379=1020.235,93.525,389.055,167.237,51.652,159.522
C04380=1020.241,93.775,389.037,167.240,51.645,159.522
C04381=1020.246,94.024,389.019,167.243,51.638,159.521
C04382=1020.251,94.273,389.001,167.245,51.632,159.520
C04383=1020.257,94.522,388.984,167.248,51.626,159.519
C04384=1020.262,94.772,388.965,167.251,51.619,159.519
C04385=1020.268,95.021,388.948,167.254,51.613,159.518
C04386=1020.273,95.270,388.930,167.256,51.606,159.517
C04387=1020.279,95.519,388.913,167.259,51.599,159.516
C04388=1020.284,95.769,388.894,167.262,51.593,159.516
C04389=1020.290,96.018,388.876,167.264,51.587,159.515
C04390=1020.295,96.267,388.858,167.268,51.580,159.514
C04391=1020.301,96.517,388.840,167.270,51.574,159.513
C04392=1020.306,96.766,388.822,167.273,51.567,159.512
C04393=1020.312,97.015,388.804,167.276,51.560,159.512
C04394=1020.317,97.264,388.787,167.278,51.554,159.511
C04395=1020.323,97.514,388.768,167.281,51.548,159.510
C04396=1020.328,97.763,388.751,167.284,51.541,159.509
C04397=1020.334,98.012,388.733,167.286,51.534,159.508
C04398=1020.339,98.262,388.715,167.289,51.528,159.508
C04399=1020.345,98.511,388.697,167.292,51.521,159.507
C04400=1020.350,98.760,388.680,167.295,51.515,159.506
C04401=1020.356,99.010,388.660,167.297,51.508,159.505
C04402=1020.361,99.259,388.643,167.301,51.502,159.505
C04403=1020.367,99.508,388.625,167.303,51.495,159.504
C04404=1020.372,99.758,388.607,167.306,51.489,159.503
C04405=1020.377,100.007,388.589,167.309,51.482,159.502
C04406=1020.383,100.256,388.570,167.311,51.476,159.502
C04407=1020.388,100.506,388.552,167.314,51.470,159.501
C04408=1020.394,100.755,388.534,167.316,51.463,159.500
C04409=1020.399,101.004,388.515,167.320,51.457,159.500
C04410=1020.405,101.253,388.497,167.322,51.450,159.499
C04411=1020.410,101.503,388.479,167.325,51.444,159.498
C04412=1020.415,101.752,388.460,167.329,51.438,159.497
C04413=1020.421,102.001,388.442,167.331,51.431,159.496
C04414=1020.426,102.250,388.424,167.334,51.425,159.496
C04415=1020.432,102.500,388.406,167.337,51.418,159.495
C04416=1020.437,102.749,388.387,167.339,51.412,159.494
C04417=1020.442,102.998,388.369,167.342,51.406,159.493
C04418=1020.448,103.247,388.351,167.344,51.399,159.493
C04419=1020.453,103.497,388.332,167.348,51.392,159.492
C04420=1020.459,103.746,388.314,167.350,51.386,159.491
C04421=1020.464,103.995,388.296,167.353,51.380,159.490
C04422=1020.470,104.244,388.278,167.356,51.373,159.490
C04423=1020.475,104.494,388.260,167.359,51.367,159.489
C04424=1020.480,104.743,388.241,167.361,51.360,159.488
C04425=1020.486,104.993,388.223,167.365,51.354,159.487
C04426=1020.491,105.242,388.204,167.367,51.347,159.487
C04427=1020.497,105.491,388.186,167.369,51.341,159.486
C04428=1020.502,105.741,388.168,167.373,51.335,159.485
C04429=1020.507,105.989,388.149,167.375,51.328,159.484
C04430=1020.513,106.239,388.131,167.378,51.321,159.483
C04431=1020.519,106.488,388.112,167.381,51.315,159.483
C04432=1020.525,106.738,388.094,167.384,51.309,159.482
C04433=1020.530,107.020,388.073,167.387,51.301,159.481
C04434=1020.536,107.303,388.052,167.390,51.294,159.480
C04435=1020.543,107.586,388.031,167.393,51.287,159.479
C04436=1020.549,107.870,388.011,167.397,51.279,159.478
C04437=1020.554,108.118,387.992,167.400,51.273,159.478
C04438=1020.560,108.368,387.974,167.402,51.266,159.477
C04439=1020.565,108.617,387.955,167.405,51.259,159.476
C04440=1020.572,108.866,387.937,167.408,51.253,159.475
C04441=1020.577,109.115,387.918,167.411,51.247,159.475
C04442=1020.582,109.365,387.900,167.414,51.240,159.474
C04443=1020.588,109.614,387.881,167.416,51.233,159.473
C04444=1020.593,109.864,387.863,167.420,51.227,159.472
C04445=1020.598,110.112,387.844,167.422,51.221,159.472
C04446=1020.604,110.362,387.825,167.425,51.214,159.471
C04447=1020.609,110.611,387.807,167.428,51.208,159.470
C04448=1020.615,110.860,387.788,167.431,51.201,159.469
C04449=1020.620,111.109,387.769,167.433,51.195,159.468
C04450=1020.626,111.359,387.750,167.437,51.188,159.468
C04451=1020.631,111.608,387.732,167.439,51.182,159.467
C04452=1020.637,111.858,387.714,167.442,51.175,159.466
C04453=1020.642,112.106,387.695,167.445,51.169,159.466
C04454=1020.648,112.356,387.675,167.448,51.163,159.465
C04455=1020.653,112.605,387.657,167.450,51.156,159.464
C04456=1020.658,112.855,387.638,167.454,51.150,159.463
C04457=1020.663,113.103,387.619,167.456,51.143,159.462
C04458=1020.669,113.353,387.600,167.459,51.137,159.462
C04459=1020.674,113.601,387.581,167.462,51.131,159.461
C04460=1020.680,113.851,387.562,167.465,51.125,159.460
C04461=1020.684,114.100,387.544,167.467,51.118,159.459
C04462=1020.690,114.350,387.524,167.471,51.112,159.459
C04463=1020.694,114.599,387.505,167.474,51.105,159.458
C04464=1020.700,114.848,387.486,167.476,51.100,159.457
C04465=1020.705,115.097,387.467,167.479,51.093,159.456
C04466=1020.711,115.346,387.448,167.482,51.087,159.456
C04467=1020.716,115.595,387.429,167.485,51.080,159.455
C04468=1020.721,115.845,387.410,167.488,51.074,159.454
C04469=1020.727,116.095,387.391,167.491,51.068,159.454
C04470=1020.732,116.343,387.372,167.493,51.061,159.453
C04471=1020.738,116.593,387.353,167.496,51.055,159.452
C04472=1020.743,116.841,387.334,167.500,51.048,159.451
C04473=1020.749,117.091,387.315,167.502,51.042,159.451
C04474=1020.754,117.340,387.296,167.505,51.036,159.450
C04475=1020.759,117.589,387.277,167.508,51.029,159.449
C04476=1020.764,117.839,387.257,167.511,51.023,159.448
C04477=1020.769,118.088,387.238,167.513,51.017,159.447
C04478=1020.775,118.338,387.219,167.517,51.011,159.447
C04479=1020.780,118.586,387.200,167.519,51.004,159.446
C04480=1020.786,118.836,387.181,167.523,50.997,159.445
C04481=1020.791,119.085,387.162,167.525,50.991,159.445
C04482=1020.796,119.334,387.143,167.528,50.985,159.444
C04483=1020.802,119.583,387.124,167.532,50.979,159.443
C04484=1020.807,119.832,387.105,167.534,50.972,159.442
C04485=1020.813,120.081,387.086,167.536,50.966,159.441
C04486=1020.819,120.331,387.066,167.540,50.959,159.441
C04487=1020.824,120.580,387.048,167.543,50.953,159.440
C04488=1020.829,120.829,387.028,167.546,50.946,159.439
C04489=1020.834,121.079,387.009,167.549,50.940,159.439
C04490=1020.839,121.328,386.990,167.551,50.934,159.438
C04491=1020.845,121.577,386.970,167.555,50.927,159.437
C04492=1020.851,121.826,386.951,167.557,50.921,159.436
C04493=1020.856,122.075,386.932,167.561,50.914,159.436
C04494=1020.861,122.325,386.913,167.564,50.908,159.435
C04495=1020.867,122.574,386.894,167.566,50.902,159.434
C04496=1020.873,122.822,386.874,167.569,50.895,159.433
C04497=1020.878,123.106,386.853,167.573,50.888,159.432
C04498=1020.884,123.389,386.831,167.576,50.881,159.432
C04499=1020.891,123.672,386.809,167.579,50.874,159.431
C04500=1020.897,123.955,386.787,167.583,50.866,159.430
C04501=1020.903,124.203,386.768,167.586,50.859,159.429
C04502=1020.908,124.452,386.748,167.588,50.853,159.428
C04503=1020.913,124.702,386.729,167.592,50.847,159.428
C04504=1020.919,124.952,386.709,167.594,50.840,159.427
C04505=1020.924,125.200,386.691,167.598,50.833,159.426
C04506=1020.930,125.450,386.671,167.600,50.827,159.425
C04507=1020.936,125.699,386.652,167.604,50.821,159.425
C04508=1020.941,125.948,386.633,167.606,50.814,159.424
C04509=1020.947,126.197,386.613,167.610,50.808,159.423
C04510=1020.952,126.446,386.594,167.612,50.801,159.422
C04511=1020.958,126.696,386.575,167.616,50.795,159.421
C04512=1020.963,126.944,386.556,167.619,50.789,159.421
C04513=1020.968,127.194,386.536,167.622,50.782,159.420
C04514=1020.974,127.444,386.517,167.625,50.775,159.419
C04515=1020.980,127.692,386.497,167.628,50.769,159.418
C04516=1020.985,127.942,386.478,167.631,50.763,159.418
C04517=1020.991,128.191,386.459,167.634,50.756,159.417
C04518=1020.996,128.440,386.439,167.637,50.750,159.416
C04519=1021.002,128.689,386.420,167.640,50.743,159.415
C04520=1021.008,128.938,386.400,167.643,50.737,159.415
C04521=1021.013,129.187,386.381,167.646,50.730,159.414
C04522=1021.018,129.437,386.362,167.649,50.724,159.413
C04523=1021.024,129.686,386.342,167.652,50.717,159.412
C04524=1021.030,129.935,386.322,167.655,50.711,159.412
C04525=1021.035,130.184,386.303,167.657,50.704,159.411
C04526=1021.040,130.433,386.284,167.661,50.698,159.410
C04527=1021.046,130.682,386.264,167.664,50.692,159.409
C04528=1021.051,130.932,386.244,167.667,50.685,159.409
C04529=1021.057,131.181,386.224,167.670,50.679,159.408
C04530=1021.062,131.430,386.205,167.673,50.672,159.407
C04531=1021.067,131.679,386.184,167.676,50.667,159.406
C04532=1021.073,131.928,386.165,167.680,50.660,159.406
C04533=1021.078,132.177,386.145,167.682,50.654,159.405
C04534=1021.084,132.427,386.125,167.685,50.648,159.404
C04535=1021.089,132.676,386.106,167.688,50.641,159.403
C04536=1021.094,132.924,386.086,167.691,50.635,159.403
C04537=1021.099,133.174,386.066,167.695,50.628,159.402
C04538=1021.105,133.423,386.046,167.697,50.622,159.401
C04539=1021.110,133.673,386.026,167.701,50.616,159.401
C04540=1021.116,133.922,386.006,167.703,50.609,159.400
C04541=1021.121,134.171,385.987,167.707,50.603,159.399
C04542=1021.127,134.420,385.967,167.710,50.596,159.398
C04543=1021.132,134.669,385.948,167.713,50.590,159.398
C04544=1021.137,134.918,385.927,167.716,50.584,159.397
C04545=1021.143,135.167,385.907,167.719,50.577,159.396
C04546=1021.148,135.417,385.887,167.722,50.571,159.395
C04547=1021.154,135.665,385.867,167.726,50.565,159.395
C04548=1021.159,135.915,385.848,167.728,50.558,159.394
C04549=1021.165,136.164,385.828,167.732,50.552,159.393
C04550=1021.170,136.414,385.808,167.734,50.545,159.392
C04551=1021.175,136.662,385.788,167.737,50.540,159.392
C04552=1021.181,136.911,385.768,167.741,50.533,159.391
C04553=1021.186,137.160,385.748,167.743,50.527,159.390
C04554=1021.192,137.409,385.728,167.747,50.520,159.389
C04555=1021.197,137.659,385.707,167.749,50.514,159.389
C04556=1021.202,137.908,385.688,167.753,50.508,159.388
C04557=1021.208,138.157,385.667,167.756,50.501,159.387
C04558=1021.214,138.406,385.647,167.759,50.495,159.387
C04559=1021.219,138.656,385.628,167.762,50.489,159.386
C04560=1021.224,138.905,385.607,167.766,50.483,159.385
C04561=1021.230,139.187,385.584,167.769,50.475,159.384
C04562=1021.236,139.470,385.561,167.772,50.468,159.383
C04563=1021.242,139.753,385.539,167.776,50.461,159.383
C04564=1021.248,140.036,385.516,167.780,50.454,159.382
C04565=1021.254,140.285,385.496,167.782,50.447,159.381
C04566=1021.259,140.534,385.475,167.786,50.441,159.380
C04567=1021.264,140.783,385.454,167.789,50.435,159.380
C04568=1021.269,141.033,385.435,167.793,50.429,159.379
C04569=1021.275,141.282,385.415,167.795,50.422,159.378
C04570=1021.280,141.531,385.394,167.799,50.416,159.378
C04571=1021.286,141.780,385.374,167.801,50.410,159.377
C04572=1021.291,142.029,385.353,167.805,50.404,159.376
C04573=1021.297,142.278,385.333,167.808,50.397,159.375
C04574=1021.302,142.528,385.313,167.812,50.391,159.375
C04575=1021.307,142.777,385.293,167.814,50.385,159.374
C04576=1021.313,143.026,385.273,167.818,50.379,159.373
C04577=1021.318,143.275,385.252,167.820,50.372,159.372
C04578=1021.324,143.524,385.232,167.824,50.365,159.372
C04579=1021.329,143.773,385.211,167.827,50.360,159.371
C04580=1021.335,144.022,385.191,167.830,50.353,159.370
C04581=1021.340,144.271,385.171,167.834,50.347,159.370
C04582=1021.345,144.520,385.150,167.837,50.340,159.369
C04583=1021.351,144.769,385.129,167.840,50.334,159.368
C04584=1021.356,145.019,385.110,167.843,50.328,159.367
C04585=1021.362,145.268,385.090,167.846,50.321,159.367
C04586=1021.367,145.517,385.069,167.849,50.315,159.366
C04587=1021.372,145.766,385.049,167.853,50.309,159.365
C04588=1021.378,146.015,385.029,167.856,50.303,159.364
C04589=1021.383,146.264,385.008,167.859,50.296,159.364
C04590=1021.389,146.513,384.987,167.863,50.290,159.363
C04591=1021.394,146.762,384.967,167.865,50.284,159.362
C04592=1021.399,147.011,384.946,167.869,50.278,159.362
C04593=1021.405,147.260,384.925,167.872,50.271,159.361
C04594=1021.411,147.510,384.904,167.876,50.265,159.360
C04595=1021.416,147.759,384.884,167.878,50.259,159.359
C04596=1021.421,148.008,384.863,167.882,50.253,159.359
C04597=1021.426,148.257,384.843,167.885,50.247,159.358
C04598=1021.432,148.506,384.822,167.888,50.240,159.357
C04599=1021.437,148.755,384.801,167.891,50.234,159.357
C04600=1021.442,149.004,384.781,167.895,50.228,159.356
C04601=1021.448,149.253,384.760,167.898,50.222,159.355
C04602=1021.453,149.502,384.739,167.901,50.215,159.355
C04603=1021.458,149.751,384.718,167.905,50.209,159.354
C04604=1021.463,150.000,384.698,167.908,50.203,159.353
C04605=1021.469,150.250,384.677,167.911,50.197,159.353
C04606=1021.475,150.498,384.656,167.914,50.190,159.352
C04607=1021.480,150.748,384.635,167.918,50.184,159.351
C04608=1021.485,150.997,384.615,167.920,50.178,159.350
C04609=1021.491,151.246,384.594,167.924,50.172,159.350
C04610=1021.496,151.495,384.574,167.928,50.165,159.349
C04611=1021.501,151.743,384.552,167.931,50.159,159.348
C04612=1021.507,151.993,384.532,167.935,50.153,159.348
C04613=1021.513,152.242,384.511,167.937,50.147,159.347
C04614=1021.518,152.492,384.490,167.941,50.141,159.346
C04615=1021.523,152.740,384.469,167.944,50.134,159.345
C04616=1021.529,152.989,384.448,167.947,50.128,159.345
C04617=1021.534,153.238,384.428,167.951,50.122,159.344
C04618=1021.539,153.487,384.407,167.954,50.116,159.343
C04619=1021.545,153.737,384.386,167.957,50.109,159.343
C04620=1021.551,153.986,384.365,167.960,50.104,159.342
C04621=1021.555,154.235,384.343,167.964,50.097,159.341
C04622=1021.561,154.484,384.323,167.968,50.091,159.341
C04623=1021.566,154.732,384.301,167.970,50.085,159.340
C04624=1021.572,154.982,384.280,167.974,50.078,159.339
C04625=1021.578,155.264,384.257,167.977,50.072,159.338
C04626=1021.584,155.547,384.233,167.982,50.065,159.338
C04627=1021.590,155.829,384.209,167.985,50.057,159.337
C04628=1021.596,156.113,384.185,167.989,50.050,159.336
C04629=1021.601,156.361,384.164,167.993,50.044,159.335
C04630=1021.607,156.610,384.143,167.996,50.038,159.335
C04631=1021.613,156.860,384.122,167.999,50.032,159.334
C04632=1021.617,157.109,384.101,168.003,50.026,159.333
C04633=1021.623,157.357,384.079,168.006,50.020,159.332
C04634=1021.628,157.607,384.059,168.009,50.014,159.332
C04635=1021.634,157.855,384.038,168.013,50.007,159.331
C04636=1021.640,158.105,384.017,168.016,50.001,159.330
C04637=1021.645,158.353,383.995,168.019,49.994,159.330
C04638=1021.650,158.603,383.974,168.023,49.988,159.329
C04639=1021.656,158.852,383.953,168.026,49.983,159.328
C04640=1021.661,159.101,383.932,168.030,49.976,159.328
C04641=1021.666,159.350,383.910,168.033,49.970,159.327
C04642=1021.672,159.599,383.889,168.037,49.964,159.326
C04643=1021.677,159.848,383.867,168.039,49.959,159.326
C04644=1021.681,160.097,383.846,168.043,49.952,159.325
C04645=1021.687,160.346,383.824,168.047,49.946,159.324
C04646=1021.692,160.595,383.802,168.050,49.940,159.324
C04647=1021.697,160.844,383.780,168.054,49.934,159.323
C04648=1021.703,161.093,383.759,168.057,49.929,159.322
C04649=1021.707,161.342,383.738,168.061,49.923,159.322
C04650=1021.712,161.591,383.716,168.063,49.916,159.321
C04651=1021.718,161.840,383.694,168.067,49.910,159.320
C04652=1021.723,162.089,383.672,168.071,49.904,159.320
C04653=1021.729,162.338,383.651,168.074,49.899,159.319
C04654=1021.734,162.586,383.629,168.078,49.893,159.319
C04655=1021.739,162.837,383.608,168.080,49.886,159.318
C04656=1021.744,163.085,383.586,168.084,49.880,159.317
C04657=1021.749,163.334,383.565,168.088,49.874,159.317
C04658=1021.755,163.583,383.542,168.091,49.868,159.316
C04659=1021.760,163.832,383.521,168.095,49.862,159.315
C04660=1021.765,164.081,383.499,168.098,49.856,159.314
C04661=1021.770,164.330,383.477,168.102,49.850,159.314
C04662=1021.776,164.579,383.456,168.105,49.844,159.313
C04663=1021.780,164.828,383.435,168.108,49.838,159.313
C04664=1021.787,165.077,383.413,168.112,49.832,159.312
C04665=1021.791,165.326,383.391,168.116,49.826,159.311
C04666=1021.796,165.575,383.369,168.119,49.820,159.311
C04667=1021.802,165.824,383.348,168.123,49.814,159.310
C04668=1021.807,166.073,383.326,168.126,49.808,159.309
C04669=1021.813,166.323,383.303,168.129,49.802,159.309
C04670=1021.818,166.571,383.282,168.133,49.796,159.308
C04671=1021.823,166.820,383.260,168.136,49.790,159.307
C04672=1021.828,167.069,383.238,168.140,49.784,159.307
C04673=1021.834,167.318,383.217,168.144,49.778,159.306
C04674=1021.839,167.567,383.195,168.146,49.772,159.305
C04675=1021.844,167.816,383.173,168.150,49.766,159.305
C04676=1021.850,168.065,383.151,168.154,49.760,159.304
C04677=1021.855,168.314,383.129,168.157,49.754,159.304
C04678=1021.860,168.563,383.107,168.161,49.748,159.303
C04679=1021.866,168.812,383.086,168.165,49.742,159.302
C04680=1021.871,169.061,383.064,168.169,49.736,159.302
C04681=1021.876,169.311,383.042,168.172,49.730,159.301
C04682=1021.882,169.559,383.020,168.176,49.724,159.300
C04683=1021.887,169.807,382.998,168.179,49.717,159.300
C04684=1021.893,170.057,382.976,168.182,49.712,159.299
C04685=1021.898,170.305,382.954,168.186,49.706,159.298
C04686=1021.904,170.555,382.932,168.190,49.700,159.298
C04687=1021.908,170.804,382.910,168.194,49.693,159.297
C04688=1021.915,171.053,382.889,168.197,49.687,159.296
C04689=1021.921,171.335,382.863,168.201,49.680,159.296
C04690=1021.926,171.617,382.839,168.205,49.674,159.295
C04691=1021.933,171.899,382.814,168.209,49.667,159.294
C04692=1021.939,172.182,382.789,168.213,49.660,159.293
C04693=1021.945,172.430,382.767,168.217,49.654,159.293
C04694=1021.950,172.680,382.745,168.221,49.648,159.292
C04695=1021.955,172.929,382.723,168.224,49.642,159.291
C04696=1021.961,173.178,382.701,168.228,49.636,159.291
C04697=1021.966,173.427,382.679,168.231,49.630,159.290
C04698=1021.972,173.675,382.656,168.235,49.624,159.290
C04699=1021.978,173.925,382.635,168.239,49.617,159.289
C04700=1021.983,174.173,382.613,168.243,49.611,159.288
C04701=1021.988,174.423,382.591,168.246,49.606,159.288
C04702=1021.993,174.671,382.568,168.250,49.600,159.287
C04703=1021.999,174.920,382.546,168.253,49.593,159.286
C04704=1022.005,175.170,382.524,168.257,49.587,159.286
C04705=1022.010,175.419,382.502,168.261,49.581,159.285
C04706=1022.016,175.667,382.480,168.265,49.575,159.284
C04707=1022.021,175.916,382.458,168.268,49.570,159.284
C04708=1022.026,176.166,382.436,168.272,49.563,159.283
C04709=1022.033,176.414,382.414,168.276,49.557,159.282
C04710=1022.038,176.663,382.392,168.280,49.551,159.282
C04711=1022.043,176.913,382.369,168.284,49.545,159.281
C04712=1022.049,177.160,382.347,168.287,49.539,159.280
C04713=1022.054,177.410,382.325,168.290,49.533,159.280
C04714=1022.060,177.660,382.303,168.294,49.527,159.279
C04715=1022.066,177.907,382.281,168.298,49.521,159.279
C04716=1022.071,178.157,382.259,168.302,49.515,159.278
C04717=1022.076,178.406,382.237,168.306,49.509,159.277
C04718=1022.082,178.654,382.215,168.310,49.503,159.277
C04719=1022.088,178.904,382.192,168.314,49.497,159.276
C04720=1022.093,179.153,382.169,168.318,49.491,159.275
C04721=1022.099,179.402,382.147,168.321,49.485,159.275
C04722=1022.105,179.650,382.125,168.324,49.479,159.274
C04723=1022.110,179.900,382.103,168.328,49.473,159.273
C04724=1022.116,180.149,382.081,168.332,49.467,159.273
C04725=1022.121,180.397,382.059,168.336,49.461,159.272
C04726=1022.127,180.647,382.037,168.340,49.454,159.272
C04727=1022.133,180.895,382.014,168.344,49.448,159.271
C04728=1022.139,181.145,381.992,168.348,49.442,159.270
C04729=1022.144,181.393,381.969,168.352,49.436,159.270
C04730=1022.149,181.642,381.947,168.356,49.430,159.269
C04731=1022.155,181.891,381.924,168.359,49.424,159.268
C04732=1022.161,182.140,381.903,168.362,49.418,159.268
C04733=1022.166,182.389,381.880,168.366,49.412,159.267
C04734=1022.171,182.638,381.856,168.370,49.406,159.267
C04735=1022.177,182.887,381.834,168.374,49.400,159.266
C04736=1022.183,183.136,381.811,168.378,49.395,159.265
C04737=1022.187,183.385,381.788,168.382,49.390,159.265
C04738=1022.193,183.634,381.765,168.386,49.384,159.264
C04739=1022.198,183.883,381.742,168.389,49.378,159.264
C04740=1022.203,184.132,381.719,168.393,49.372,159.263
C04741=1022.208,184.381,381.697,168.397,49.366,159.263
C04742=1022.214,184.630,381.674,168.400,49.360,159.262
C04743=1022.219,184.879,381.650,168.404,49.354,159.261
C04744=1022.225,185.128,381.627,168.408,49.348,159.261
C04745=1022.230,185.376,381.605,168.413,49.343,159.260
C04746=1022.235,185.625,381.581,168.417,49.337,159.260
C04747=1022.240,185.874,381.558,168.421,49.331,159.259
C04748=1022.246,186.123,381.535,168.424,49.326,159.258
C04749=1022.251,186.371,381.512,168.428,49.320,159.258
C04750=1022.256,186.620,381.489,168.432,49.314,159.257
C04751=1022.262,186.869,381.466,168.436,49.308,159.257
C04752=1022.267,187.118,381.443,168.440,49.302,159.256
C04753=1022.273,187.401,381.417,168.445,49.296,159.256
C04754=1022.279,187.682,381.391,168.448,49.289,159.255
C04755=1022.285,187.964,381.365,168.453,49.283,159.254
C04756=1022.291,188.245,381.338,168.457,49.277,159.253
C04757=1022.297,188.496,381.316,168.461,49.271,159.253
C04758=1022.302,188.745,381.293,168.465,49.265,159.252
C04759=1022.308,188.995,381.269,168.469,49.259,159.252
C04760=1022.313,189.246,381.246,168.473,49.253,159.251
C04761=1022.319,189.494,381.222,168.477,49.247,159.250
C04762=1022.324,189.742,381.200,168.481,49.242,159.250
C04763=1022.329,189.992,381.176,168.485,49.236,159.250
C04764=1022.335,190.240,381.153,168.489,49.230,159.249
C04765=1022.341,190.489,381.130,168.493,49.224,159.248
C04766=1022.346,190.739,381.107,168.497,49.218,159.248
C04767=1022.351,190.987,381.084,168.501,49.212,159.247
C04768=1022.357,191.236,381.061,168.505,49.207,159.247
C04769=1022.362,191.486,381.037,168.510,49.201,159.246
C04770=1022.368,191.734,381.013,168.513,49.196,159.245
C04771=1022.374,191.983,380.991,168.517,49.190,159.245
C04772=1022.378,192.231,380.967,168.521,49.184,159.244
C04773=1022.384,192.480,380.944,168.525,49.178,159.244
C04774=1022.389,192.729,380.921,168.529,49.172,159.243
C04775=1022.395,192.978,380.897,168.533,49.167,159.243
C04776=1022.401,193.226,380.874,168.537,49.161,159.242
C04777=1022.406,193.476,380.851,168.541,49.155,159.241
C04778=1022.411,193.725,380.828,168.545,49.149,159.241
C04779=1022.417,193.974,380.805,168.549,49.144,159.240
C04780=1022.422,194.222,380.781,168.553,49.138,159.240
C04781=1022.428,194.471,380.758,168.558,49.133,159.239
C04782=1022.434,194.720,380.735,168.562,49.127,159.239
C04783=1022.439,194.968,380.710,168.566,49.121,159.238
C04784=1022.445,195.217,380.687,168.570,49.115,159.237
C04785=1022.450,195.467,380.664,168.574,49.109,159.237
C04786=1022.456,195.715,380.641,168.578,49.103,159.236
C04787=1022.462,195.964,380.617,168.582,49.098,159.236
C04788=1022.467,196.213,380.594,168.586,49.092,159.235
C04789=1022.473,196.463,380.570,168.590,49.086,159.235
C04790=1022.479,196.711,380.547,168.595,49.080,159.234
C04791=1022.484,196.960,380.523,168.599,49.074,159.234
C04792=1022.490,197.208,380.500,168.603,49.069,159.233
C04793=1022.496,197.457,380.477,168.607,49.063,159.233
C04794=1022.501,197.706,380.453,168.611,49.057,159.232
C04795=1022.507,197.955,380.429,168.615,49.051,159.231
C04796=1022.512,198.204,380.406,168.619,49.046,159.231
C04797=1022.518,198.452,380.382,168.624,49.040,159.230
C04798=1022.524,198.701,380.359,168.628,49.035,159.230
C04799=1022.529,198.950,380.335,168.632,49.029,159.229
C04800=1022.535,199.199,380.312,168.636,49.023,159.229
C04801=1022.541,199.448,380.288,168.640,49.018,159.228
C04802=1022.546,199.697,380.265,168.644,49.012,159.228
C04803=1022.552,199.945,380.240,168.649,49.006,159.227
C04804=1022.557,200.194,380.217,168.653,49.000,159.226
C04805=1022.563,200.443,380.193,168.658,48.995,159.226
C04806=1022.568,200.691,380.169,168.662,48.989,159.225
C04807=1022.573,200.941,380.145,168.666,48.984,159.225
C04808=1022.579,201.190,380.121,168.670,48.978,159.224
C04809=1022.585,201.438,380.097,168.675,48.973,159.224
C04810=1022.590,201.687,380.073,168.679,48.967,159.223
C04811=1022.595,201.936,380.049,168.683,48.961,159.223
C04812=1022.601,202.184,380.026,168.687,48.956,159.222
C04813=1022.607,202.434,380.001,168.691,48.950,159.222
C04814=1022.612,202.683,379.977,168.695,48.945,159.221
C04815=1022.617,202.931,379.953,168.699,48.939,159.221
C04816=1022.623,203.180,379.929,168.703,48.933,159.220
C04817=1022.651,204.420,379.808,169.131,49.027,159.304
C04818=1022.657,204.630,379.787,169.135,49.023,159.304
C04819=1022.662,204.842,379.765,169.137,49.019,159.304
C04820=1022.668,205.053,379.744,169.139,49.014,159.303
C04821=1022.673,205.264,379.722,169.142,49.010,159.303
C04822=1022.679,205.475,379.700,169.145,49.007,159.302
C04823=1022.684,205.686,379.678,169.148,49.002,159.302
C04824=1022.689,205.898,379.657,169.151,48.998,159.301
C04825=1022.696,206.146,379.630,169.155,48.994,159.301
C04826=1022.702,206.395,379.605,169.158,48.989,159.301
C04827=1022.709,206.644,379.579,169.160,48.985,159.300
C04828=1022.715,206.892,379.553,169.164,48.981,159.300
C04829=1022.721,207.140,379.528,169.167,48.976,159.299
C04830=1022.728,207.389,379.503,169.171,48.971,159.298
C04831=1022.735,207.638,379.476,169.174,48.967,159.298
C04832=1022.741,207.887,379.451,169.178,48.962,159.298
C04833=1022.747,208.135,379.425,169.181,48.957,159.297
C04834=1022.753,208.384,379.399,169.185,48.953,159.297
C04835=1022.759,208.632,379.374,169.188,48.948,159.296
C04836=1022.766,208.881,379.347,169.192,48.944,159.296
C04837=1022.772,209.130,379.322,169.194,48.939,159.295
C04838=1022.779,209.378,379.296,169.197,48.935,159.295
C04839=1022.785,209.626,379.270,169.201,48.930,159.294
C04840=1022.792,209.875,379.244,169.204,48.925,159.294
C04841=1022.798,210.124,379.218,169.208,48.921,159.293
C04842=1022.804,210.372,379.192,169.211,48.916,159.293
C04843=1022.810,210.621,379.167,169.215,48.912,159.293
C04844=1022.816,210.869,379.140,169.218,48.907,159.292
C04845=1022.823,211.118,379.114,169.221,48.904,159.292
C04846=1022.829,211.367,379.088,169.224,48.899,159.291
C04847=1022.835,211.615,379.062,169.228,48.895,159.291
C04848=1022.841,211.864,379.036,169.232,48.890,159.290
C04849=1022.849,212.112,379.010,169.235,48.886,159.290
C04850=1022.854,212.361,378.983,169.239,48.881,159.290
C04851=1022.861,212.609,378.958,169.242,48.877,159.289
C04852=1022.867,212.857,378.932,169.245,48.873,159.289
C04853=1022.873,213.106,378.905,169.249,48.869,159.288
C04854=1022.880,213.355,378.880,169.252,48.864,159.288
C04855=1022.886,213.603,378.853,169.256,48.859,159.287
C04856=1022.892,213.852,378.826,169.259,48.855,159.287
C04857=1022.899,214.101,378.801,169.263,48.850,159.286
C04858=1022.905,214.349,378.775,169.266,48.846,159.286
C04859=1022.911,214.597,378.748,169.269,48.842,159.286
C04860=1022.918,214.847,378.723,169.272,48.838,159.285
C04861=1022.924,215.095,378.697,169.276,48.833,159.285
C04862=1022.930,215.343,378.670,169.279,48.829,159.284
C04863=1022.937,215.592,378.644,169.283,48.824,159.284
C04864=1022.943,215.841,378.618,169.287,48.820,159.284
C04865=1022.950,216.090,378.591,169.290,48.815,159.283
C04866=1022.956,216.338,378.565,169.293,48.812,159.283
C04867=1022.962,216.586,378.539,169.296,48.807,159.282
C04868=1022.969,216.835,378.512,169.300,48.803,159.282
C04869=1022.975,217.083,378.487,169.303,48.798,159.281
C04870=1022.981,217.332,378.460,169.307,48.794,159.281
C04871=1022.988,217.581,378.434,169.311,48.790,159.281
C04872=1022.995,217.829,378.408,169.314,48.785,159.280
C04873=1023.001,218.078,378.381,169.317,48.781,159.280
C04874=1023.008,218.326,378.355,169.321,48.777,159.279
C04875=1023.014,218.574,378.329,169.324,48.773,159.279
C04876=1023.020,218.823,378.302,169.328,48.769,159.279
C04877=1023.026,219.036,378.279,169.331,48.765,159.278
C04878=1023.031,219.248,378.257,169.334,48.762,159.278
C04879=1023.036,219.460,378.234,169.336,48.758,159.278
C04880=1023.041,219.674,378.211,169.339,48.755,159.277
C04881=1023.047,219.886,378.188,169.343,48.751,159.277
C04882=1023.052,220.099,378.166,169.346,48.748,159.277
C04883=1023.058,220.311,378.143,169.349,48.744,159.276
C04884=1023.063,220.524,378.120,169.352,48.741,159.276
C04885=1023.069,220.773,378.094,169.355,48.736,159.276
C04886=1023.076,221.021,378.066,169.359,48.732,159.275
C04887=1023.082,221.269,378.040,169.362,48.728,159.275
C04888=1023.089,221.518,378.013,169.365,48.724,159.274
C04889=1023.095,221.766,377.987,169.369,48.719,159.274
C04890=1023.101,222.016,377.960,169.373,48.715,159.274
C04891=1023.108,222.264,377.934,169.376,48.711,159.273
C04892=1023.113,222.512,377.907,169.379,48.707,159.273
C04893=1023.120,222.761,377.880,169.383,48.703,159.273
C04894=1023.126,223.009,377.854,169.386,48.699,159.272
C04895=1023.133,223.258,377.827,169.390,48.695,159.272
C04896=1023.139,223.506,377.799,169.394,48.691,159.272
C04897=1023.146,223.755,377.773,169.396,48.687,159.271
C04898=1023.152,224.003,377.746,169.400,48.683,159.271
C04899=1023.158,224.252,377.719,169.404,48.679,159.271
C04900=1023.164,224.500,377.693,169.408,48.675,159.270
C04901=1023.171,224.748,377.666,169.411,48.671,159.270
C04902=1023.177,224.997,377.639,169.415,48.667,159.270
C04903=1023.184,225.246,377.612,169.418,48.663,159.269
C04904=1023.190,225.495,377.585,169.422,48.659,159.269
C04905=1023.197,225.743,377.559,169.425,48.655,159.268
C04906=1023.204,225.991,377.532,169.429,48.650,159.268
C04907=1023.209,226.240,377.505,169.433,48.646,159.268
C04908=1023.216,226.488,377.479,169.436,48.642,159.267
C04909=1023.222,226.737,377.452,169.439,48.638,159.267
C04910=1023.229,226.985,377.424,169.443,48.635,159.267
C04911=1023.235,227.233,377.398,169.447,48.631,159.266
C04912=1023.241,227.482,377.370,169.450,48.627,159.266
C04913=1023.248,227.730,377.344,169.454,48.622,159.266
C04914=1023.254,227.979,377.317,169.457,48.619,159.265
C04915=1023.261,228.227,377.289,169.461,48.615,159.265
C04916=1023.267,228.476,377.262,169.465,48.611,159.265
C04917=1023.273,228.724,377.235,169.468,48.607,159.264
C04918=1023.279,228.973,377.208,169.471,48.604,159.264
C04919=1023.286,229.221,377.180,169.475,48.600,159.264
C04920=1023.292,229.469,377.154,169.479,48.595,159.263
C04921=1023.298,229.718,377.126,169.482,48.591,159.263
C04922=1023.305,229.967,377.099,169.486,48.588,159.263
C04923=1023.310,230.215,377.072,169.489,48.584,159.263
C04924=1023.318,230.463,377.045,169.493,48.580,159.262
C04925=1023.324,230.712,377.017,169.497,48.576,159.262
C04926=1023.330,230.960,376.990,169.501,48.572,159.262
C04927=1023.336,231.209,376.962,169.504,48.569,159.261
C04928=1023.342,231.457,376.936,169.507,48.565,159.261
C04929=1023.349,231.706,376.908,169.511,48.561,159.261
C04930=1023.355,231.954,376.880,169.515,48.557,159.261
C04931=1023.361,232.203,376.854,169.519,48.553,159.260
C04932=1023.368,232.451,376.826,169.522,48.550,159.260
C04933=1023.375,232.699,376.798,169.526,48.546,159.260
C04934=1023.380,232.948,376.772,169.530,48.542,159.259
C04935=1023.387,233.196,376.744,169.533,48.538,159.259
C04936=1023.394,233.445,376.716,169.536,48.535,159.259
C04937=1023.403,233.862,376.670,169.542,48.529,159.258
C04938=1023.414,234.279,376.624,169.548,48.523,159.258
C04939=1023.426,234.697,376.578,169.555,48.516,159.257
C04940=1023.435,235.114,376.532,169.561,48.510,159.257
C04941=1023.442,235.363,376.504,169.565,48.506,159.257
C04942=1023.449,235.611,376.476,169.568,48.502,159.256
C04943=1023.455,235.860,376.450,169.572,48.499,159.256
C04944=1023.461,236.108,376.422,169.576,48.495,159.256
C04945=1023.468,236.356,376.394,169.579,48.492,159.256
C04946=1023.475,236.605,376.366,169.583,48.487,159.255
C04947=1023.481,236.853,376.339,169.587,48.484,159.255
C04948=1023.487,237.101,376.311,169.591,48.480,159.255
C04949=1023.494,237.350,376.284,169.594,48.477,159.254
C04950=1023.500,237.599,376.256,169.598,48.473,159.254
C04951=1023.506,237.847,376.229,169.601,48.469,159.254
C04952=1023.512,238.095,376.201,169.605,48.466,159.254
C04953=1023.519,238.344,376.173,169.610,48.462,159.254
C04954=1023.526,238.592,376.145,169.612,48.458,159.253
C04955=1023.532,238.840,376.118,169.616,48.455,159.253
C04956=1023.538,239.088,376.090,169.620,48.451,159.253
C04957=1023.544,239.337,376.062,169.624,48.447,159.252
C04958=1023.551,239.585,376.034,169.628,48.444,159.252
C04959=1023.558,239.834,376.007,169.631,48.441,159.252
C04960=1023.564,240.083,375.978,169.635,48.437,159.252
C04961=1023.570,240.330,375.951,169.639,48.433,159.251
C04962=1023.577,240.579,375.923,169.642,48.430,159.251
C04963=1023.582,240.827,375.895,169.646,48.427,159.251
C04964=1023.589,241.076,375.867,169.650,48.423,159.251
C04965=1023.595,241.325,375.839,169.654,48.420,159.251
C04966=1023.602,241.572,375.810,169.657,48.417,159.250
C04967=1023.608,241.820,375.783,169.661,48.412,159.250
C04968=1023.614,242.069,375.755,169.665,48.409,159.250
C04969=1023.621,242.317,375.727,169.669,48.405,159.250
C04970=1023.627,242.566,375.699,169.672,48.402,159.250
C04971=1023.633,242.815,375.671,169.676,48.399,159.249
C04972=1023.640,243.062,375.642,169.680,48.395,159.249
C04973=1023.646,243.310,375.614,169.684,48.392,159.249
C04974=1023.652,243.559,375.587,169.687,48.389,159.249
C04975=1023.658,243.808,375.558,169.691,48.385,159.248
C04976=1023.665,244.055,375.530,169.695,48.382,159.248
C04977=1023.671,244.304,375.502,169.699,48.379,159.248
C04978=1023.678,244.552,375.473,169.702,48.375,159.248
C04979=1023.684,244.801,375.444,169.706,48.372,159.248
C04980=1023.690,245.049,375.417,169.710,48.368,159.248
C04981=1023.696,245.297,375.388,169.714,48.365,159.247
C04982=1023.702,245.546,375.360,169.718,48.362,159.247
C04983=1023.709,245.794,375.331,169.722,48.358,159.247
C04984=1023.715,246.042,375.303,169.726,48.355,159.247
C04985=1023.721,246.290,375.274,169.729,48.352,159.247
C04986=1023.728,246.539,375.246,169.733,48.348,159.246
C04987=1023.734,246.788,375.218,169.737,48.345,159.246
C04988=1023.740,247.036,375.189,169.740,48.342,159.246
C04989=1023.747,247.284,375.161,169.744,48.339,159.246
C04990=1023.753,247.532,375.132,169.748,48.336,159.246
C04991=1023.759,247.781,375.104,169.752,48.332,159.246
C04992=1023.765,248.029,375.075,169.755,48.329,159.245
C04993=1023.775,248.440,375.027,169.762,48.323,159.245
C04994=1023.786,248.851,374.980,169.769,48.318,159.245
C04995=1023.796,249.262,374.933,169.775,48.313,159.245
C04996=1023.807,249.674,374.886,169.781,48.307,159.244
C04997=1023.814,249.922,374.857,169.785,48.305,159.244
C04998=1023.820,250.171,374.829,169.789,48.301,159.244
C04999=1023.827,250.418,374.800,169.793,48.298,159.244
C05000=1023.833,250.667,374.771,169.797,48.294,159.244
C05001=1023.839,250.915,374.743,169.800,48.291,159.243
C05002=1023.845,251.163,374.714,169.804,48.288,159.243
C05003=1023.852,251.411,374.685,169.808,48.285,159.243
C05004=1023.858,251.660,374.657,169.813,48.282,159.243
C05005=1023.864,251.908,374.628,169.816,48.279,159.243
C05006=1023.871,252.156,374.600,169.820,48.276,159.243
C05007=1023.877,252.405,374.571,169.824,48.272,159.243
C05008=1023.883,252.653,374.542,169.828,48.269,159.243
C05009=1023.890,252.901,374.513,169.831,48.266,159.242
C05010=1023.897,253.149,374.485,169.835,48.263,159.242
C05011=1023.903,253.398,374.456,169.840,48.259,159.242
C05012=1023.909,253.646,374.427,169.844,48.257,159.242
C05013=1023.916,253.894,374.399,169.847,48.254,159.242
C05014=1023.923,254.142,374.369,169.851,48.250,159.242
C05015=1023.929,254.391,374.341,169.855,48.247,159.242
C05016=1023.935,254.639,374.312,169.859,48.244,159.242
C05017=1023.942,254.887,374.284,169.864,48.240,159.241
C05018=1023.948,255.135,374.255,169.867,48.238,159.241
C05019=1023.955,255.384,374.225,169.871,48.235,159.241
C05020=1023.962,255.632,374.197,169.875,48.231,159.241
C05021=1023.968,255.880,374.168,169.879,48.228,159.241
C05022=1023.974,256.129,374.139,169.882,48.225,159.241
C05023=1023.980,256.377,374.110,169.887,48.222,159.241
C05024=1023.988,256.625,374.082,169.891,48.219,159.240
C05025=1023.994,256.874,374.053,169.895,48.216,159.240
C05026=1024.000,257.122,374.023,169.899,48.213,159.240
C05027=1024.007,257.370,373.994,169.902,48.210,159.240
C05028=1024.014,257.618,373.966,169.907,48.207,159.240
C05029=1024.021,257.866,373.937,169.911,48.204,159.240
C05030=1024.027,258.115,373.908,169.915,48.201,159.240
C05031=1024.033,258.363,373.879,169.919,48.197,159.240
C05032=1024.040,258.611,373.850,169.923,48.195,159.240
C05033=1024.047,258.859,373.821,169.927,48.191,159.239
C05034=1024.053,259.107,373.792,169.931,48.189,159.239
C05035=1024.060,259.355,373.763,169.935,48.185,159.239
C05036=1024.067,259.604,373.734,169.940,48.182,159.239
C05037=1024.073,259.852,373.705,169.943,48.179,159.239
C05038=1024.079,260.100,373.676,169.947,48.177,159.239
C05039=1024.086,260.348,373.647,169.951,48.173,159.239
C05040=1024.093,260.597,373.618,169.955,48.170,159.239
C05041=1024.100,260.845,373.588,169.960,48.168,159.239
C05042=1024.106,261.093,373.559,169.963,48.164,159.239
C05043=1024.112,261.341,373.529,169.967,48.162,159.239
C05044=1024.119,261.589,373.499,169.972,48.159,159.239
C05045=1024.125,261.837,373.470,169.976,48.156,159.239
C05046=1024.131,262.086,373.441,169.979,48.153,159.238
C05047=1024.138,262.333,373.411,169.984,48.150,159.238
C05048=1024.145,262.582,373.382,169.988,48.148,159.238
C05049=1024.155,262.992,373.333,169.995,48.143,159.238
C05050=1024.165,263.401,373.285,170.001,48.139,159.238
C05051=1024.176,263.811,373.236,170.008,48.134,159.238
C05052=1024.187,264.221,373.187,170.014,48.129,159.238
C05053=1024.193,264.468,373.158,170.019,48.126,159.238
C05054=1024.200,264.717,373.128,170.023,48.123,159.238
C05055=1024.207,264.964,373.098,170.027,48.120,159.238
C05056=1024.212,265.213,373.069,170.031,48.118,159.238
C05057=1024.219,265.461,373.039,170.035,48.115,159.238
C05058=1024.226,265.709,373.010,170.040,48.112,159.238
C05059=1024.232,265.957,372.980,170.044,48.110,159.238
C05060=1024.239,266.206,372.950,170.047,48.107,159.238
C05061=1024.245,266.453,372.920,170.051,48.104,159.238
C05062=1024.252,266.702,372.890,170.056,48.101,159.238
C05063=1024.258,266.950,372.861,170.060,48.098,159.238
C05064=1024.264,267.198,372.831,170.064,48.096,159.237
C05065=1024.271,267.446,372.801,170.068,48.093,159.237
C05066=1024.278,267.694,372.771,170.072,48.090,159.237
C05067=1024.285,267.942,372.741,170.077,48.088,159.237
C05068=1024.290,268.191,372.712,170.081,48.085,159.237
C05069=1024.297,268.439,372.682,170.085,48.082,159.237
C05070=1024.304,268.686,372.652,170.089,48.080,159.237
C05071=1024.310,268.935,372.622,170.094,48.077,159.238
C05072=1024.317,269.183,372.592,170.098,48.075,159.238
C05073=1024.323,269.430,372.562,170.101,48.072,159.237
C05074=1024.330,269.679,372.532,170.106,48.069,159.237
C05075=1024.336,269.927,372.503,170.110,48.067,159.237
C05076=1024.343,270.175,372.472,170.115,48.064,159.237
C05077=1024.349,270.423,372.442,170.119,48.061,159.237
C05078=1024.356,270.671,372.412,170.122,48.059,159.237
C05079=1024.362,270.919,372.382,170.127,48.057,159.238
C05080=1024.369,271.167,372.351,170.132,48.054,159.238
C05081=1024.375,271.415,372.321,170.136,48.051,159.238
C05082=1024.382,271.663,372.291,170.139,48.049,159.238
C05083=1024.388,271.911,372.261,170.144,48.046,159.237
C05084=1024.395,272.160,372.231,170.148,48.044,159.238
C05085=1024.401,272.409,372.201,170.153,48.041,159.238
C05086=1024.408,272.656,372.171,170.157,48.038,159.238
C05087=1024.414,272.905,372.140,170.161,48.036,159.238
C05088=1024.421,273.152,372.110,170.165,48.034,159.238
C05089=1024.427,273.401,372.080,170.170,48.031,159.238
C05090=1024.434,273.648,372.050,170.174,48.028,159.238
C05091=1024.440,273.897,372.019,170.178,48.026,159.238
C05092=1024.446,274.144,371.988,170.182,48.024,159.238
C05093=1024.453,274.392,371.958,170.187,48.021,159.238
C05094=1024.460,274.641,371.927,170.191,48.019,159.238
C05095=1024.466,274.888,371.897,170.196,48.016,159.238
C05096=1024.473,275.137,371.867,170.199,48.014,159.238
C05097=1024.480,275.385,371.837,170.204,48.012,159.238
C05098=1024.486,275.633,371.806,170.208,48.009,159.238
C05099=1024.492,275.881,371.776,170.213,48.006,159.238
C05100=1024.499,276.128,371.745,170.217,48.004,159.238
C05101=1024.505,276.377,371.714,170.221,48.001,159.238
C05102=1024.512,276.625,371.684,170.225,47.999,159.238
C05103=1024.518,276.873,371.654,170.230,47.997,159.238
C05104=1024.525,277.121,371.624,170.234,47.994,159.238
C05105=1024.536,277.535,371.572,170.242,47.990,159.239
C05106=1024.547,277.949,371.520,170.249,47.987,159.239
C05107=1024.558,278.363,371.469,170.256,47.982,159.239
C05108=1024.569,278.778,371.418,170.264,47.979,159.239
C05109=1024.574,279.026,371.387,170.268,47.976,159.239
C05110=1024.582,279.274,371.356,170.272,47.974,159.239
C05111=1024.588,279.522,371.326,170.276,47.972,159.239
C05112=1024.594,279.769,371.295,170.281,47.969,159.239
C05113=1024.601,280.018,371.264,170.286,47.967,159.240
C05114=1024.608,280.266,371.232,170.290,47.965,159.240
C05115=1024.614,280.514,371.202,170.294,47.963,159.240
C05116=1024.621,280.761,371.171,170.298,47.961,159.240
C05117=1024.627,281.010,371.140,170.303,47.958,159.240
C05118=1024.634,281.257,371.109,170.307,47.956,159.240
C05119=1024.640,281.506,371.078,170.312,47.954,159.240
C05120=1024.647,281.754,371.047,170.316,47.952,159.240
C05121=1024.653,282.002,371.017,170.320,47.949,159.240
C05122=1024.660,282.249,370.986,170.325,47.947,159.240
C05123=1024.667,282.497,370.954,170.330,47.945,159.241
C05124=1024.674,282.746,370.924,170.334,47.943,159.241
C05125=1024.680,282.994,370.892,170.339,47.940,159.241
C05126=1024.686,283.241,370.862,170.343,47.938,159.241
C05127=1024.693,283.489,370.830,170.347,47.936,159.241
C05128=1024.700,283.737,370.799,170.352,47.934,159.241
C05129=1024.707,283.986,370.769,170.356,47.931,159.241
C05130=1024.713,284.233,370.737,170.361,47.929,159.241
C05131=1024.720,284.481,370.706,170.366,47.927,159.242
C05132=1024.727,284.729,370.674,170.370,47.925,159.242
C05133=1024.733,284.977,370.644,170.374,47.923,159.242
C05134=1024.739,285.225,370.613,170.379,47.921,159.242
C05135=1024.747,285.473,370.582,170.383,47.918,159.242
C05136=1024.754,285.720,370.550,170.388,47.916,159.242
C05137=1024.760,285.969,370.518,170.393,47.914,159.242
C05138=1024.766,286.217,370.488,170.398,47.912,159.243
C05139=1024.773,286.465,370.456,170.401,47.910,159.243
C05140=1024.779,286.713,370.425,170.406,47.908,159.243
C05141=1024.786,286.961,370.393,170.411,47.906,159.243
C05142=1024.793,287.209,370.362,170.415,47.904,159.243
C05143=1024.800,287.457,370.331,170.420,47.902,159.243
C05144=1024.806,287.704,370.299,170.425,47.900,159.243
C05145=1024.813,287.952,370.268,170.429,47.898,159.244
C05146=1024.819,288.200,370.237,170.433,47.896,159.244
C05147=1024.826,288.448,370.205,170.438,47.894,159.244
C05148=1024.833,288.695,370.174,170.443,47.892,159.244
C05149=1024.839,288.944,370.142,170.447,47.890,159.244
C05150=1024.845,289.192,370.110,170.452,47.888,159.244
C05151=1024.852,289.440,370.079,170.457,47.886,159.245
C05152=1024.859,289.687,370.047,170.461,47.884,159.245
C05153=1024.866,289.935,370.015,170.466,47.882,159.245
C05154=1024.873,290.183,369.984,170.470,47.880,159.245
C05155=1024.879,290.431,369.952,170.475,47.878,159.245
C05156=1024.885,290.679,369.920,170.480,47.876,159.246
C05157=1024.892,290.927,369.889,170.484,47.874,159.246
C05158=1024.899,291.174,369.857,170.490,47.872,159.246
C05159=1024.906,291.422,369.825,170.494,47.870,159.246
C05160=1024.913,291.670,369.794,170.498,47.869,159.246
C05161=1024.918,291.884,369.766,170.503,47.866,159.247
C05162=1024.924,292.097,369.739,170.507,47.865,159.247
C05163=1024.930,292.309,369.712,170.510,47.863,159.247
C05164=1024.935,292.523,369.684,170.514,47.862,159.247
C05165=1024.942,292.736,369.656,170.518,47.861,159.247
C05166=1024.947,292.950,369.630,170.523,47.858,159.248
C05167=1024.953,293.163,369.602,170.527,47.857,159.248
C05168=1024.959,293.376,369.574,170.531,47.855,159.248
C05169=1024.965,293.624,369.542,170.535,47.853,159.248
C05170=1024.972,293.872,369.511,170.540,47.852,159.248
C05171=1024.979,294.119,369.478,170.545,47.850,159.249
C05172=1024.985,294.367,369.446,170.550,47.848,159.249
C05173=1024.991,294.615,369.414,170.554,47.847,159.249
C05174=1024.998,294.862,369.382,170.559,47.845,159.249
C05175=1025.004,295.111,369.350,170.564,47.843,159.250
C05176=1025.011,295.358,369.317,170.569,47.842,159.250
C05177=1025.018,295.606,369.285,170.573,47.840,159.250
C05178=1025.024,295.854,369.252,170.578,47.838,159.250
C05179=1025.031,296.102,369.220,170.583,47.836,159.251
C05180=1025.037,296.349,369.187,170.587,47.835,159.251
C05181=1025.043,296.598,369.155,170.592,47.833,159.251
C05182=1025.050,296.845,369.123,170.597,47.831,159.251
C05183=1025.057,297.092,369.090,170.602,47.830,159.252
C05184=1025.063,297.341,369.058,170.607,47.828,159.252
C05185=1025.070,297.589,369.026,170.612,47.826,159.252
C05186=1025.077,297.836,368.993,170.616,47.824,159.252
C05187=1025.084,298.083,368.961,170.622,47.823,159.253
C05188=1025.090,298.331,368.928,170.626,47.822,159.253
C05189=1025.097,298.580,368.896,170.630,47.820,159.253
C05190=1025.104,298.827,368.864,170.635,47.818,159.254
C05191=1025.110,299.075,368.831,170.640,47.817,159.254
C05192=1025.116,299.322,368.798,170.645,47.815,159.254
C05193=1025.124,299.570,368.766,170.650,47.813,159.255
C05194=1025.130,299.818,368.733,170.655,47.812,159.255
C05195=1025.136,300.066,368.700,170.660,47.810,159.255
C05196=1025.143,300.314,368.669,170.665,47.808,159.255
C05197=1025.150,300.562,368.636,170.670,47.807,159.256
C05198=1025.157,300.809,368.604,170.675,47.805,159.256
C05199=1025.163,301.057,368.571,170.680,47.803,159.256
C05200=1025.170,301.305,368.538,170.685,47.802,159.257
C05201=1025.177,301.552,368.506,170.689,47.801,159.257
C05202=1025.184,301.800,368.473,170.694,47.799,159.257
C05203=1025.190,302.048,368.440,170.699,47.798,159.258
C05204=1025.198,302.295,368.408,170.704,47.796,159.258
C05205=1025.204,302.544,368.374,170.709,47.794,159.258
C05206=1025.211,302.791,368.342,170.714,47.793,159.258
C05207=1025.218,303.038,368.309,170.719,47.791,159.259
C05208=1025.225,303.286,368.276,170.724,47.790,159.259
C05209=1025.231,303.534,368.243,170.729,47.788,159.260
C05210=1025.239,303.782,368.210,170.734,47.787,159.260
C05211=1025.245,304.029,368.178,170.739,47.785,159.260
C05212=1025.252,304.278,368.145,170.744,47.783,159.260
C05213=1025.259,304.525,368.112,170.749,47.782,159.261
C05214=1025.266,304.772,368.079,170.754,47.780,159.261
C05215=1025.273,305.020,368.046,170.759,47.779,159.261
C05216=1025.280,305.268,368.014,170.764,47.778,159.262
C05217=1025.287,305.516,367.981,170.769,47.776,159.262
C05218=1025.293,305.763,367.948,170.774,47.775,159.263
C05219=1025.301,306.011,367.915,170.779,47.773,159.263
C05220=1025.307,306.258,367.882,170.784,47.772,159.263
C05221=1025.314,306.481,367.852,170.789,47.770,159.264
C05222=1025.320,306.702,367.823,170.793,47.769,159.264
C05223=1025.326,306.924,367.793,170.798,47.768,159.264
C05224=1025.332,307.146,367.764,170.802,47.767,159.264
C05225=1025.339,307.368,367.734,170.807,47.765,159.265
C05226=1025.345,307.590,367.705,170.811,47.764,159.265
C05227=1025.351,307.812,367.675,170.816,47.762,159.265
C05228=1025.357,308.033,367.645,170.820,47.761,159.266
C05229=1025.364,308.281,367.612,170.826,47.760,159.266
C05230=1025.372,308.529,367.579,170.831,47.759,159.267
C05231=1025.378,308.776,367.546,170.836,47.758,159.267
C05232=1025.386,309.024,367.512,170.841,47.756,159.267
C05233=1025.393,309.272,367.480,170.846,47.755,159.268
C05234=1025.400,309.519,367.446,170.852,47.753,159.268
C05235=1025.407,309.767,367.413,170.857,47.752,159.268
C05236=1025.415,310.015,367.380,170.862,47.750,159.269
C05237=1025.421,310.262,367.347,170.867,47.749,159.269
C05238=1025.428,310.510,367.314,170.872,47.748,159.270
C05239=1025.435,310.757,367.280,170.877,47.746,159.270
C05240=1025.442,311.005,367.247,170.883,47.746,159.271
C05241=1025.449,311.253,367.213,170.888,47.744,159.271
C05242=1025.455,311.500,367.179,170.893,47.743,159.271
C05243=1025.462,311.748,367.145,170.898,47.742,159.272
C05244=1025.469,311.996,367.111,170.903,47.741,159.272
C05245=1025.475,312.243,367.077,170.908,47.740,159.273
C05246=1025.482,312.491,367.044,170.914,47.739,159.273
C05247=1025.489,312.738,367.010,170.919,47.737,159.274
C05248=1025.496,312.985,366.976,170.924,47.736,159.274
C05249=1025.502,313.233,366.942,170.929,47.735,159.274
C05250=1025.510,313.481,366.908,170.935,47.734,159.275
C05251=1025.516,313.728,366.875,170.940,47.733,159.275
C05252=1025.523,313.976,366.840,170.945,47.732,159.276
C05253=1025.530,314.223,366.806,170.950,47.731,159.276
C05254=1025.537,314.471,366.773,170.955,47.730,159.277
C05255=1025.543,314.718,366.739,170.961,47.729,159.277
C05256=1025.550,314.966,366.705,170.966,47.727,159.278
C05257=1025.557,315.214,366.671,170.971,47.727,159.278
C05258=1025.564,315.461,366.637,170.976,47.726,159.279
C05259=1025.570,315.709,366.603,170.982,47.724,159.279
C05260=1025.578,315.956,366.569,170.987,47.724,159.280
C05261=1025.585,316.204,366.535,170.993,47.722,159.280
C05262=1025.592,316.451,366.500,170.998,47.721,159.280
C05263=1025.599,316.699,366.466,171.004,47.720,159.281
C05264=1025.606,316.947,366.433,171.009,47.719,159.282
C05265=1025.612,317.195,366.398,171.014,47.719,159.282
C05266=1025.619,317.441,366.364,171.019,47.717,159.282
C05267=1025.626,317.689,366.330,171.025,47.716,159.283
C05268=1025.633,317.937,366.296,171.030,47.715,159.283
C05269=1025.640,318.184,366.262,171.035,47.715,159.284
C05270=1025.648,318.431,366.227,171.041,47.713,159.284
C05271=1025.654,318.679,366.193,171.047,47.712,159.285
C05272=1025.661,318.927,366.159,171.052,47.711,159.285
C05273=1025.669,319.174,366.125,171.058,47.710,159.286
C05274=1025.675,319.422,366.090,171.063,47.710,159.287
C05275=1025.682,319.670,366.056,171.068,47.709,159.287
C05276=1025.690,319.917,366.022,171.074,47.708,159.288
C05277=1025.696,320.165,365.987,171.079,47.707,159.288
C05278=1025.704,320.412,365.953,171.085,47.705,159.289
C05279=1025.711,320.660,365.919,171.090,47.705,159.289
C05280=1025.718,320.907,365.884,171.096,47.704,159.290
C05281=1025.725,321.131,365.853,171.101,47.703,159.290
C05282=1025.731,321.356,365.822,171.105,47.702,159.291
C05283=1025.737,321.580,365.791,171.111,47.702,159.291
C05284=1025.744,321.804,365.759,171.116,47.701,159.292
C05285=1025.750,322.029,365.728,171.121,47.700,159.292
C05286=1025.756,322.253,365.697,171.126,47.699,159.293
C05287=1025.763,322.478,365.666,171.131,47.698,159.293
C05288=1025.770,322.703,365.634,171.136,47.697,159.294
C05289=1025.778,322.950,365.599,171.142,47.696,159.294
C05290=1025.784,323.198,365.565,171.147,47.696,159.295
C05291=1025.792,323.445,365.531,171.153,47.695,159.295
C05292=1025.799,323.692,365.496,171.158,47.695,159.296
C05293=1025.806,323.940,365.462,171.164,47.693,159.296
C05294=1025.814,324.188,365.427,171.170,47.693,159.297
C05295=1025.821,324.435,365.392,171.175,47.692,159.297
C05296=1025.828,324.682,365.357,171.180,47.691,159.298
C05297=1025.835,324.930,365.323,171.187,47.690,159.299
C05298=1025.843,325.177,365.289,171.192,47.689,159.299
C05299=1025.850,325.425,365.253,171.198,47.689,159.300
C05300=1025.858,325.672,365.219,171.203,47.688,159.300
C05301=1025.864,325.920,365.184,171.210,47.687,159.301
C05302=1025.872,326.168,365.149,171.215,47.686,159.301
C05303=1025.880,326.415,365.115,171.220,47.685,159.302
C05304=1025.886,326.662,365.080,171.226,47.685,159.303
C05305=1025.894,326.909,365.045,171.232,47.684,159.303
C05306=1025.902,327.157,365.010,171.238,47.683,159.304
C05307=1025.909,327.404,364.975,171.243,47.683,159.305
C05308=1025.916,327.652,364.940,171.249,47.682,159.305
C05309=1025.923,327.900,364.904,171.255,47.682,159.306
C05310=1025.930,328.147,364.870,171.261,47.681,159.306
C05311=1025.937,328.393,364.834,171.266,47.680,159.307
C05312=1025.945,328.641,364.798,171.272,47.680,159.308
C05313=1025.952,328.889,364.763,171.278,47.679,159.308
C05314=1025.958,329.136,364.728,171.284,47.678,159.309
C05315=1025.967,329.384,364.693,171.290,47.678,159.310
C05316=1025.974,329.631,364.657,171.295,47.677,159.310
C05317=1025.980,329.878,364.622,171.302,47.677,159.311
C05318=1025.988,330.126,364.587,171.307,47.676,159.312
C05319=1025.995,330.373,364.551,171.313,47.676,159.312
C05320=1026.003,330.621,364.516,171.319,47.675,159.313
C05321=1026.010,330.868,364.481,171.325,47.675,159.314
C05322=1026.017,331.115,364.445,171.330,47.674,159.314
C05323=1026.024,331.363,364.410,171.336,47.674,159.315
C05324=1026.031,331.610,364.374,171.342,47.673,159.316
C05325=1026.039,331.857,364.339,171.348,47.673,159.316
C05326=1026.046,332.105,364.304,171.354,47.673,159.317
C05327=1026.054,332.352,364.267,171.360,47.672,159.318
C05328=1026.061,332.600,364.232,171.366,47.671,159.318
C05329=1026.068,332.847,364.196,171.371,47.671,159.319
C05330=1026.075,333.094,364.161,171.378,47.671,159.320
C05331=1026.083,333.341,364.125,171.383,47.670,159.320
C05332=1026.090,333.588,364.090,171.389,47.670,159.321
C05333=1026.098,333.836,364.054,171.396,47.669,159.322
C05334=1026.105,334.084,364.018,171.401,47.669,159.323
C05335=1026.113,334.330,363.982,171.407,47.669,159.323
C05336=1026.120,334.579,363.946,171.414,47.668,159.324
C05337=1026.126,334.826,363.910,171.420,47.668,159.325
C05338=1026.134,335.073,363.874,171.425,47.668,159.325
C05339=1026.141,335.320,363.838,171.432,47.667,159.326
C05340=1026.149,335.567,363.802,171.438,47.667,159.327
C05341=1026.155,335.790,363.770,171.443,47.666,159.327
C05342=1026.162,336.012,363.737,171.449,47.666,159.328
C05343=1026.169,336.234,363.705,171.454,47.666,159.329
C05344=1026.175,336.456,363.672,171.459,47.666,159.330
C05345=1026.182,336.679,363.641,171.465,47.666,159.330
C05346=1026.188,336.901,363.608,171.470,47.666,159.331
C05347=1026.195,337.123,363.576,171.476,47.665,159.331
C05348=1026.202,337.345,363.543,171.481,47.665,159.332
C05349=1026.209,337.592,363.507,171.487,47.664,159.333
C05350=1026.217,337.839,363.471,171.494,47.664,159.334
C05351=1026.224,338.087,363.435,171.500,47.664,159.335
C05352=1026.232,338.334,363.398,171.505,47.664,159.335
C05353=1026.239,338.581,363.363,171.512,47.663,159.336
C05354=1026.247,338.828,363.326,171.518,47.663,159.337
C05355=1026.254,339.076,363.290,171.525,47.663,159.338
C05356=1026.261,339.323,363.253,171.530,47.663,159.338
C05357=1026.269,339.570,363.216,171.537,47.663,159.339
C05358=1026.276,339.817,363.181,171.543,47.662,159.340
C05359=1026.284,340.064,363.144,171.550,47.663,159.341
C05360=1026.292,340.312,363.108,171.555,47.662,159.342
C05361=1026.299,340.560,363.071,171.561,47.662,159.342
C05362=1026.307,340.806,363.034,171.568,47.662,159.343
C05363=1026.314,341.053,362.998,171.574,47.662,159.344
C05364=1026.322,341.300,362.962,171.581,47.662,159.345
C05365=1026.329,341.548,362.925,171.586,47.662,159.346
C05366=1026.336,341.795,362.889,171.593,47.661,159.347
C05367=1026.344,342.042,362.852,171.599,47.662,159.347
C05368=1026.351,342.290,362.815,171.606,47.661,159.348
C05369=1026.359,342.537,362.778,171.612,47.662,159.349
C05370=1026.366,342.784,362.741,171.618,47.661,159.350
C05371=1026.374,343.031,362.704,171.624,47.662,159.351
C05372=1026.382,343.279,362.668,171.631,47.662,159.352
C05373=1026.388,343.525,362.631,171.637,47.662,159.352
C05374=1026.396,343.772,362.595,171.644,47.662,159.353
C05375=1026.404,344.019,362.558,171.650,47.661,159.354
C05376=1026.411,344.266,362.520,171.657,47.662,159.355
C05377=1026.419,344.514,362.484,171.663,47.662,159.356
C05378=1026.426,344.761,362.446,171.669,47.661,159.357
C05379=1026.434,345.008,362.409,171.675,47.662,159.358
C05380=1026.441,345.256,362.373,171.682,47.662,159.359
C05381=1026.450,345.503,362.335,171.688,47.662,159.360
C05382=1026.458,345.750,362.298,171.695,47.662,159.360
C05383=1026.465,345.997,362.261,171.702,47.662,159.361
C05384=1026.473,346.244,362.224,171.708,47.662,159.362
C05385=1026.480,346.492,362.187,171.715,47.662,159.363
C05386=1026.488,346.739,362.150,171.721,47.663,159.364
C05387=1026.495,346.986,362.113,171.728,47.662,159.365
C05388=1026.503,347.232,362.076,171.735,47.662,159.366
C05389=1026.510,347.480,362.038,171.741,47.663,159.367
C05390=1026.519,347.727,362.001,171.748,47.663,159.368
C05391=1026.527,347.974,361.964,171.754,47.663,159.369
C05392=1026.534,348.221,361.926,171.761,47.663,159.370
C05393=1026.541,348.468,361.889,171.768,47.664,159.371
C05394=1026.549,348.715,361.852,171.774,47.664,159.371
C05395=1026.557,348.962,361.814,171.781,47.664,159.372
C05396=1026.564,349.210,361.777,171.787,47.664,159.373
C05397=1026.573,349.456,361.739,171.794,47.665,159.374
C05398=1026.580,349.703,361.701,171.801,47.665,159.375
C05399=1026.587,349.950,361.664,171.807,47.665,159.376
C05400=1026.595,350.197,361.627,171.814,47.666,159.377
C05401=1026.602,350.418,361.593,171.820,47.666,159.378
C05402=1026.609,350.638,361.559,171.826,47.666,159.379
C05403=1026.616,350.859,361.525,171.832,47.666,159.380
C05404=1026.622,351.080,361.492,171.838,47.667,159.381
C05405=1026.630,351.301,361.458,171.844,47.667,159.382
C05406=1026.636,351.521,361.424,171.850,47.667,159.383
C05407=1026.644,351.742,361.391,171.856,47.668,159.383
C05408=1026.650,351.962,361.357,171.863,47.668,159.384
C05409=1026.658,352.210,361.319,171.869,47.668,159.385
C05410=1026.667,352.456,361.281,171.876,47.668,159.386
C05411=1026.674,352.704,361.243,171.883,47.669,159.387
C05412=1026.682,352.950,361.205,171.889,47.669,159.388
C05413=1026.690,353.197,361.168,171.896,47.670,159.389
C05414=1026.698,353.444,361.130,171.903,47.670,159.390
C05415=1026.705,353.691,361.092,171.910,47.670,159.391
C05416=1026.714,353.938,361.054,171.916,47.671,159.392
C05417=1026.722,354.185,361.016,171.924,47.671,159.393
C05418=1026.730,354.433,360.978,171.931,47.672,159.394
C05419=1026.737,354.679,360.940,171.938,47.672,159.396
C05420=1026.746,354.926,360.902,171.944,47.673,159.396
C05421=1026.753,355.173,360.864,171.951,47.673,159.398
C05422=1026.761,355.420,360.825,171.959,47.674,159.399
C05423=1026.769,355.667,360.787,171.966,47.674,159.400
C05424=1026.777,355.914,360.749,171.972,47.675,159.401
C05425=1026.785,356.161,360.710,171.979,47.675,159.402
C05426=1026.793,356.408,360.672,171.986,47.676,159.403
C05427=1026.800,356.654,360.634,171.994,47.677,159.404
C05428=1026.809,356.902,360.595,172.001,47.677,159.405
C05429=1026.816,357.149,360.557,172.008,47.677,159.406
C05430=1026.824,357.396,360.519,172.014,47.678,159.407
C05431=1026.833,357.643,360.481,172.022,47.679,159.409
C05432=1026.841,357.889,360.442,172.029,47.680,159.410
C05433=1026.849,358.136,360.403,172.036,47.680,159.411
C05434=1026.857,358.383,360.365,172.043,47.680,159.412
C05435=1026.865,358.630,360.326,172.051,47.681,159.413
C05436=1026.873,358.877,360.288,172.057,47.682,159.414
C05437=1026.881,359.124,360.249,172.064,47.683,159.415
C05438=1026.888,359.371,360.211,172.072,47.684,159.416
C05439=1026.897,359.617,360.172,172.079,47.684,159.418
C05440=1026.905,359.864,360.133,172.086,47.685,159.419
C05441=1026.913,360.111,360.095,172.094,47.686,159.420
C05442=1026.921,360.358,360.056,172.101,47.686,159.421
C05443=1026.929,360.605,360.017,172.108,47.687,159.422
C05444=1026.937,360.852,359.978,172.116,47.688,159.423
C05445=1026.944,361.098,359.939,172.123,47.688,159.424
C05446=1026.953,361.345,359.900,172.129,47.689,159.426
C05447=1026.961,361.592,359.861,172.137,47.690,159.427
C05448=1026.969,361.839,359.822,172.144,47.691,159.428
C05449=1026.977,362.086,359.782,172.152,47.692,159.429
C05450=1026.985,362.332,359.743,172.159,47.693,159.430
C05451=1026.993,362.579,359.705,172.166,47.693,159.432
C05452=1027.001,362.826,359.665,172.174,47.695,159.433
C05453=1027.009,363.073,359.626,172.181,47.695,159.434
C05454=1027.017,363.320,359.587,172.189,47.696,159.435
